(* Logix 5000 project; controller cal1615 1756-L62 rev 20.19; software revision 20.05; part 5 of 81 *)

        [6]   // Zone 1 Dint to HMI
        [6].0   // Zone 1 Dint to HMI Exhaut VFD Faulted
        [6].1   // Zone 1 Dint to HMI Exhaut VFD Warning
        [6].2   // Zone 1 Dint to HMI Exhaut VFD Running Forward
        [6].3   // Zone 1 Dint to HMI Exhaut VFD Running Reverse
        [6].4   // Zone 1 Dint to HMI Exhaut VFD Ready
        [6].5   // Zone 1 Dint to HMI Exhaut VFD Control from Net
        [6].6   // Zone 1 Dint to HMI Exhaut VFD Reference from Net
        [6].7   // Zone 1 Dint to HMI Exhaut VFD at Reference
        [6].8   // Zone 1 Dint to HMI Recirc VFD Faulted
        [6].9   // Zone 1 Dint to HMI Recirc VFD Warning
        [6].10   // Zone 1 Dint to HMI Recirc VFD Running Forward
        [6].11   // Zone 1 Dint to HMI Recirc VFD Running Reverse
        [6].12   // Zone 1 Dint to HMI Recirc VFD Ready
        [6].13   // Zone 1 Dint to HMI Recirc VFD Control from Net
        [6].14   // Zone 1 Dint to HMI Recirc VFD Reference from Net
        [6].15   // Zone 1 Dint to HMI Recirc VFD At Reference
        [6].16   // Zone 1 Dint to HMI Temperature Control PI: Request Heat
        [6].17   // Zone 1 Dint to HMI Temperature Control PI: Off
        [6].18   // Zone 1 Dint to HMI Temperature Control PI: Request Manual Control
        [6].19   // Zone 1 Dint to HMI Temperature Control PI:
        [6].20   // Zone 1 Dint to HMI PI:
        [6].21   // Zone 1 Dint to HMI PI:
        [6].22   // Zone 1 Dint to HMI PI:
        [6].23   // Zone 1 Dint to HMI PI:
        [6].24   // Zone 1 Dint to HMI PI:
        [6].25   // Zone 1 Dint to HMI PI:
        [6].26   // Zone 1 Dint to HMI PI:
        [6].27   // Zone 1 Dint to HMI PI:
        [6].28   // Zone 1 Dint to HMI PI:
        [6].29   // Zone 1 Dint to HMI PI:
        [6].30   // Zone 1 Dint to HMI PI:
        [6].31   // Zone 1 Dint to HMI PI:
        [7]   // Zone 1 Dint to HMI
        [8]   // Zone 1 Dint to HMI Temperature Control Status - State
        [9]   // Zone 1 Dint to HMI Temperature Control Status (Ready/Fault etc)
        [10]   // Zone 1 Dint to HMI Exhaust VFD Status
        [11]   // Zone 1 Dint to HMI Recirc VFD Status
        [12]   // Zone 1 Dint to HMI
        [13]   // Zone 1 Dint to HMI
        [14]   // Zone 1 Dint to HMI
        [15]   // Zone 1 Dint to HMI
   p11_do_enable_burner : BOOL := 1;   // Zone 1 Digital Output Enable Burner
   p11_do_exh : acs800_do_normal := (forward := 1);   // Zone 1 Digital Output Exhaust Fan
   p11_do_recirc : acs800_do_normal := (forward := 1);   // Zone 1 Digital Outputs Supply Fan
   p11_do_rst_flame : BOOL;   // Zone 1 Digital Output Reset Flame Safety
   p11_exhaust_input_max : REAL := 2000.0;
   p11_exhaust_input_min : REAL;   // Zone 1 Exhaust Input Minimum
   p11_exhaust_output_max : REAL := 2000.0;
   p11_exhaust_output_min : REAL;
   p11_hc_input_max : REAL := 100.0;
   p11_hc_input_min : REAL;
   p11_hc_output_max : REAL := 30840.0;
   p11_hc_output_min : REAL;
   p11_lfl_input_max : REAL := 30840.0;
   p11_lfl_input_min : REAL;
   p11_lfl_output_max : REAL := 100.0;
   p11_lfl_output_min : REAL;
   p11_param_fast_to_soak : REAL := 20.0;   // Zone 1 Parameter Fast to Soak Control
   p11_param_lfl_hhl : REAL := 40.0;   // Zone 1 Parameter High High Lower Flash Limit
   p11_param_lfl_hl : REAL := 25.0;   // Zone 1 Parameter High LFL Limit
   p11_param_pid1_ff : REAL := 25.0;   // Zone 1 Parameter Fast PID Bias
   p11_param_pid1_kd : REAL;   // Zone 1 Parameter Fast PID Derivative Gain
   p11_param_pid1_ki : REAL;   // Zone 1 Parameter Fast PID Integral Gain
   p11_param_pid1_kp : REAL := 50.0;   // Zone 1 Parameter Fast PID Proportional Gain
   p11_param_pid2_ff : REAL := 20.0;   // Zone 1 Parameter Auto PID Bias
   p11_param_pid2_kd : REAL;   // Zone 1 Parameter Auto PID Derivative Gain
   p11_param_pid2_ki : REAL := 1.0;   // Zone 1 Parameter Auto PID Integral Gain
   p11_param_pid2_kp : REAL := 20.0;   // Zone 1 Parameter Auto PID Proportional Gain
   p11_param_shutdown_temp : REAL := 110.0;   // Zone 1 Parameter Zone Shutdown Temperature
   p11_param_soak_to_fast : REAL := 20.0;   // Zone 1 Parameter Soak to Fast Control
   p11_param_tc01_dev : REAL := 20.0;   // Zone 1 Parameter Oven Temperature Deviation from Setpoint
   p11_param_tc01_hl : REAL := 440.0;   // Zone 1 Parameter Process Air High Limit
   p11_param_tc01z : REAL;   // Zone 1 Parameter Process Temperature Zero Offset
   p11_param_tc02z : REAL;   // Zone 1 Parameter SupplyTemperature Zero Offset
   p11_param_zone_pressure : REAL := -0.25;   // Zone 1 Parameter High Pressure LImit
   p11_prs_input_max : REAL := 30840.0;
   p11_prs_input_min : REAL;
   p11_prs_output_max : REAL := 0.25;
   p11_prs_output_min : REAL := -0.25;
   p11_real_to_hmi : REAL[112] := ([0] := 194.7, [1] := 194.7, [2] := 194.7, [6] := -0.25, [7] := 3.0804152, [8] := 30.891432, [9] := 4.9, [10] := 901.0, [12] := 37.748573, [13] := 22.2, [14] := 1101.0, [24] := 17.754694, [28] := 900.0, [30] := 1100.0, [44] := 50.0, [47] := 25.0, [48] := 20.0, [49] := 1.0, [51] := 20.0, [52] := 440.0, [54] := 20.0, [55] := 25.0, [56] := 40.0, [57] := 110.0, [58] := -0.25, [59] := 20.0, [60] := 20.0, [67] := 195.0, [68] := 45.0, [72] := 194.7);   // Zone 1 Real to HMI
        [0]   // Zone 1 Real to HMI Analog Input Zone 1 Process Control Temperature 1
        [1]   // Zone 1 Real to HMI Analog Input Zone 1 Process Control Temperature 2
        [2]   // Zone 1 Real to HMI Analog Input
        [3]   // Zone 1 Real to HMI Analog Input
        [6]   // Zone 1 Real to HMI Analog Input Pressure
        [7]   // Zone 1 Real to HMI Analog Input Lower Flash Limit
        [8]   // Zone 1 Real to HMI Analog Input Exhaust Fan Hz
        [9]   // Zone 1 Real to HMI Analog Input Exhaust Fan Amps
        [10]   // Zone 1 Real to HMI Analog Input Exhaust Fan RPM
        [11]   // Zone 1 Real to HMI Analog Input Exhaust Fan PCT
        [12]   // Zone 1 Real to HMI Analog Input Recirc Fan Hz
        [13]   // Zone 1 Real to HMI Analog Input Recirc Fan Amps
        [14]   // Zone 1 Real to HMI Analog Analog Input Recirc Fan RPM
        [15]   // Zone 1 Real to HMI Analog Analog Input Recirc Fan Pct
        [16]   // Zone 1 Real to HMI Analog Input Spare
        [17]   // Zone 1 Real to HMI Analog Input Spare
        [24]   // Zone 1 Real to HMI Analog Output Hot Air Damper
        [28]   // Zone 1 Real to HMI Analog Output Exhaust Fan VFD Selected Speed
        [30]   // Zone 1 Real to HMI Analog Output Supply Fan VFD Selected Speed
        [40]   // Zone 1 Real to HMI Parameter TC01 Temperature Zero Offset
        [41]   // Zone 1 Real to HMI Parameter TC02 Temperature Zero Offset
        [42]   // Zone 1 Real to HMI Parameter
        [43]   // Zone 1 Real to HMI Parameter
        [44]   // Zone 1 Real to HMI Parameter PID1 NKp
        [45]   // Zone 1 Real to HMI Parameter PID1 Ki
        [46]   // Zone 1 Real to HMI Parameter PID1 Kd
        [47]   // Zone 1 Real to HMI Parameter PID1 Bias
        [48]   // Zone 1 Real to HMI Parameter PID2 Kp
        [49]   // Zone 1 Real to HMI Parameter PID2 Ki
        [50]   // Zone 1 Real to HMI Parameter PID2 Kd
        [51]   // Zone 1 Real to HMI Parameter PID2 Bias
        [52]   // Zone 1 Real to HMI Parameter Process Control High Limit
        [53]   // Zone 1 Real to HMI Parameter Spare
        [54]   // Zone 1 Real to HMI parameter Process Control Deviation
        [55]   // Zone 1 Real to HMI Parameter LFL Warning Level
        [56]   // Zone 1 Real to HMI Parameter LFL Alarm Level
        [57]   // Zone 1 Real to HMI Parameter Zone Shutdown Temperature
        [58]   // Zone 1 Real to HMI Parameter High Pressure LImit
        [59]   // Zone 1 Real to HMI Temperature Control Fast to Soak Control Deviation
        [60]   // Zone 1 Real to HMI Temperature Control Soak to Fast Control Deviation
        [61]   // Zone 1 Real to HMI Parameter
        [62]   // Zone 1 Real to HMI Parameter
        [63]   // Zone 1 Real to HMI Parameter
        [64]   // Zone 1 Real to HMI Exhaust VFD RPM Setpoint
        [65]   // Zone 1 Real to HMI Recirc VFD RPM Setpoint
        [67]   // Zone 1 Real to HMI Temperature Control Setpoint
        [68]   // Zone 1 Real to HMI Temperature Control manual Control Valve Setpoint
        [69]   // Zone 1 Real to HMI
        [70]   // Zone 1 Real to HMI
        [71]   // Zone 1 Real to HMI
        [72]   // Zone 1 Real to HMI Process Control Temperature
        [73]   // Zone 1 Real to HMI
        [74]   // Zone 1 Real to HMI
        [75]   // Zone 1 Real to HMI
        [76]   // Zone 1 Real to HMI
        [77]   // Zone 1 Real to HMI
        [78]   // Zone 1 Real to HMI
        [79]   // Zone 1 Real to HMI
   p11_recirc_input_max : REAL := 2000.0;
   p11_recirc_input_min : REAL;
   p11_recirc_output_max : REAL := 2000.0;
   p11_recirc_output_min : REAL;
   p11r01 : routine := (comment := 7);   // Zone 1 Main
   p11r02 : routine := (comment := -1073741761);   // Zone 1 Misc Control
        .FAULT.0   // Zone 1 Misc Control
        .WARNING.0   // Zone 1 Misc Control Low Pressure
        .UNACK_FAULT   // Zone 1 Misc Control Unacknowledged Fault Exists
        .UNACK_WARNING   // Zone 1 Misc Control Unacknowledged Warning Exists
   p11r02_fault_exists : BOOL;
   p11r02_not_safe_temp : BOOL := 1;   // Zone 1 Misc Control Zone above Safe Temp
   p11r02_safe_temp : BOOL;   // Zone 1 Misc Control Zone Temperature at Safe Temp
   p11r02_shutdown_temp : BOOL;   // Zone 1 Misc Control Safe Shutdown Temperature
   p11r02_timer_fault : TIMER[4];   // Zone 1 Misc Control Fault Delay
   p11r02_timer_safe_temp : TIMER[2] := ([0].PRE := 30000, [1].PRE := 30000, [1].ACC := 30018, [1].EN := 1, [1].DN := 1);   // Zone 1 Misc Control Chamber SafeTemperature Dwell
   p11r02_timer_warning : TIMER[4] := ([0].PRE := 1500);   // Zone 1 Misc Control Warning Delay
   p11r02_unack_fault : BOOL;   // Zone 1 Misc Control Unacknowledged Fault Exists
   p11r02_unack_warning : BOOL;   // Zone 1 Misc Control Unacknowledged Warning Exists
   p11r02_warning_exists : BOOL := 1;
   p11r03 : routine := (comment := -1073741761);   // Zone 1 Input
        .UNACK_FAULT   // Zone 1 Input Unacknowledged Fault Exists
        .UNACK_WARNING   // Zone 1 Input Unacknowledged Warning Exists
   p11r03_hz : SYS_SCP := (Input := 901.0, Input_Max := 1750.0, Output_Max := 60.0, Output := 30.891432);   // Zone 1 Analog Inputs SCP Hz
   p11r03_timer_fault : TIMER[4];   // Zone 1 Input Fault Delay
   p11r03_timer_warning : TIMER[4];   // Zone 1 Input Warning Delay
   p11r04 : routine := (comment := -1073741761);   // Zone 1 Output
        .UNACK_FAULT   // Zone 1 Analog Output Unacknowledged Fault Exists
        .UNACK_WARNING   // Zone 1 Analog Output Unacknowledged Warning Exists
   p11r04_timer_fault : TIMER[4];   // Zone 1 Output Fault Delay
   p11r04_timer_warning : TIMER[4];   // Zone 1 Output Warning Delay
   p11r05 : routine := (comment := -1073741761, state := 7);   // Zone 1 Dint to HMI
        .UNACK_FAULT   // Zone 1 Dint to HMI Unacknowledged Fault Exists
        .UNACK_WARNING   // Zone 1 Dint to HMI Unacknowledged Warning Exists
   p11r05_exh_status : DINT := 2;
   p11r05_recirc_status : DINT := 2;
   p11r05_temp_ctrl_status : DINT := 2;
   p11r05_timer_fault : TIMER[4];   // Zone 1 Dint to HMI Fault Delay
   p11r05_timer_warning : TIMER[4];   // Zone 1 Dint to HMI Warning Delay
   p11r06 : routine := (comment := -1073741572);   // Zone 1 Real to HMI
        .UNACK_FAULT   // Zone 1 Real to HMI Unacknowledged Fault Exists
        .UNACK_WARNING   // Zone 1 Real to HMI Unacknowledged Warning Exists
   p11r06_timer_fault : TIMER[4];   // Zone 1 Real to HMI Fault Delay
   p11r06_timer_warning : TIMER[4];   // Zone 1 Real to HMI Warning Delay
   p11r07 : routine := (comment := -1073741761);   // Zone 1 Alarms
        .UNACK_FAULT   // Zone 1 Alarms Unacknowledged Fault Exists
        .UNACK_WARNING   // Zone 1 Alarms Unacknowledged Warning Exists
   p11r07_timer_fault : TIMER[4];   // Zone 1 Alarms Fault Delay
   p11r07_timer_warning : TIMER[4];   // Zone 1 Alarms Warning Delay
   p11r08 : routine := (comment := -1073741761);   // Zone 1 Warnings
        .UNACK_FAULT   // Zone 1 Warnings Unacknowledged Fault Exists
        .UNACK_WARNING   // Zone 1 Warnings Unacknowledged Warning Exists
   p11r08_timer_fault : TIMER[4];   // Zone 1 Warnings Fault Delay
   p11r08_timer_warning : TIMER[4];   // Zone 1 Warnings Warning Delay
   p11r09 : routine := (comment := -1073741761);   // Zone 1 Modes
        .FAULT.0   // Zone 1 Modes
        .UNACK_FAULT   // Zone 1 Modes Unacknowledged Fault Exists
        .UNACK_WARNING   // Zone 1 Modes Unacknowledged Warning Exists
   p11r09_timer_fault : TIMER[4];   // Zone 1 Modes Fault Delay
   p11r09_timer_warning : TIMER[8];   // Zone 1 Modes Warning Delay
   p11r10 : routine := (comment := -1073741761);   // Zone 1
        .UNACK_FAULT   // Zone 1 Parameters Unacknowledged Fault Exists
        .UNACK_WARNING   // Zone 1 Parameters Unacknowledged Warning Exists
   p11r10_timer_fault : TIMER[4];   // Zone 1 Fault Delay
   p11r10_timer_warning : TIMER[4];   // Zone 1 Warning Delay
   p11r12_Oven_auto_run_on : BOOL := 1;   // Zone 1 Temp Sequence Oven Auto Run On
   p11r16_pid_temp_cv : DINT := 16;   // Zone 1 Temperature Control Control Valve
   p11r16_temp_ok : BOOL := 1;   // Zone 1 Temperature Control Temperature OK
   p11r20 : routine := (comment := -1073741761);   // Zone 1 Temp Sequence
        .FAULT.0   // Zone 1
        .FAULT.1   // Zone 1
        .FAULT.2   // Zone 1
        .FAULT.3   // Zone 1
        .WARNING.0   // Zone 1
        .UNACK_FAULT   // Zone 1 Temp Sequence Unacknowledged Fault Exists
        .UNACK_WARNING   // Zone 1 Unacknowledged Warning Exists
   p11r20_safeties_ok : BOOL := 1;   // Zone 1 Temperature Control Burner Safeties OK this Lightoff
   p11r20_state : DINT := 1025;   // Zone 1 Temperature Control State
        .0   // Zone 1 Temperature Control State 0 One-Step per Scan
        .1   // Zone 1 Temperature Control State 1 Off
        .2   // Zone 1 Temperature Control State 2 Idle
        .3   // Zone 1 Temperature Control State 3 Start Recirculation Fan
        .4   // Zone 1 Temperature Control State 4 Start Exhaust Fan
        .5   // Zone 1 Temperature Control State 5 Wait for Safeties
        .6   // Zone 1 Temperature Control State 6 Safeties Made
        .7   // Zone 1 Temperature Control State 7 Purge
        .8   // Zone 1 Temperature Control State 8 Burner Lit
        .9   // Zone 1 Temperature Control State 9 Heat to Setpoint
        .10   // Zone 1 Temperature Control State 10 Control to Setpoint
        .11   // Zone 1 Temperature Control State 11 Cooldown
        .12   // Zone 1 Temperature Control State 12 Cooldown Fans
        .13   // Zone 1 Temperature Control State 13 Complete
        .31   // Zone 1 Temperature Control State 31 Manual
   p11r20_status : DINT := 10;   // Zone 1 Temperature Control Sequence Status
   p11r20_timer_fault : TIMER[4];   // Zone 1 Temp Sequence Fault Delay
   p11r20_timer_state_11 : TIMER := (PRE := 5000);   // Zone 1 Temp Sequence State 11 Dwell
   p11r20_timer_state_3 : TIMER := (PRE := 1000, ACC := 1022, EN := 1, DN := 1);   // Zone 1 Temperature Control State 3 Dwell
   p11r20_timer_state_4 : TIMER := (PRE := 1000, ACC := 1025, EN := 1, DN := 1);   // Zone 1 Temp Sequence State 4 Dwell
   p11r20_timer_state_7 : TIMER := (PRE := 2000, ACC := 2024, EN := 1, DN := 1);   // Zone 1 Temp Sequence State 7 Dwell
   p11r20_timer_warning : TIMER[4];   // Zone 1 Temp Sequence Warning Delay
   p11r30 : routine := (comment := -1073741697, oneshot := 4, warning := 192, warning_ack := 192);   // Zone 1 Temperature Control
        .FAULT.0   // Zone 1 Temperature Control Process Control Software High Limit
        .FAULT.1   // Zone 1 Temperature Control Process Control Hardware High Limit
        .FAULT.2   // Zone 1 Temperature Control Process Control Thermocouple Failure
        .FAULT.3   // Zone 1 Temperature Control Process Control Temperature Spare
        .FAULT.4   // Zone 1 Temperature Control Lower Flash Limit High High Limit Exceeded
        .FAULT.5   // Zone 1 Temperature Control Flame Failure
        .FAULT.6   // Zone 1 Temperature Control Burner Safeties Failure
        .FAULT.7   // Zone 1 Temperature Control Recirculation Fan Speed Fault
        .FAULT.8   // Zone 1 Temperature Control Exhaust Fan Speed Fault
        .FAULT.9   // Zone 1 Temperature Control Access Door Open
        .FAULT.10   // Zone 1 Temperature Control Spare
        .FAULT.11   // Zone 1 Temperature Control
        .FAULT.12   // Zone 1 Temperature Control Spare
        .FAULT.13   // Zone 1 Temperature Control
        .FAULT.14   // Zone 1 Temperature Control
        .WARNING.0   // Zone 1 Temperature Control Control Temperature Deviation
        .WARNING.1   // Zone 1 Temperature Control Process Control Thermocouple 1 Failure
        .WARNING.2   // Zone 1 Temperature Control Process Control Thermocouple 2 Failure
        .WARNING.3   // Zone 1 Temperature Control Control Valve in Manual
        .WARNING.4   // Zone 1 Temperature Control LFL High Limit
        .WARNING.5   // Zone 1 Temperature Control Zone Off
        .WARNING.6   // Zone 1 Temperature Control Fresh Air Filter Dirty
        .WARNING.7   // Zone 1 Temperature Control Combustion Air Filter Dirty
        .WARNING.8   // Zone 1 Temperature Control Recirculation Air Filter Dirty
        .UNACK_FAULT   // Zone 1 Temperature Control Unacknowledged Fault Exists
        .UNACK_WARNING   // Zone 1 Temperature Control Unacknowledged Warning Exists
   p11r30_cv_man_sp : REAL := 45.0;   // Zone 1 Temperature Control Manual Heat Control Valve Setpoint
   p11r30_pb_auto : BOOL;   // Zone 1 Temperature Control PB: Zone Control Auto
   p11r30_pb_manual : BOOL;   // Zone 1 Temperature Control PB: Zone Control Manual
   p11r30_pb_zone_off : BOOL;   // Zone 1 Temperature Control PB: Stop Zone Heat Control
   p11r30_pb_zone_on : BOOL;   // Zone 1 Temperature Control PB: Start Zone Heat Control
   p11r30_permissive_run : BOOL := 1;   // Zone 1 Temperature Control Run Permissive
   p11r30_pid_temp : PID := (CTL := -2144304000, EN := 1, NOBC := 1, NOZC := 1, INI := 1, DVNA := 1, PVHA := 1, SP := 195.0, KP := 20.0, KI := 1.0, BIAS := 20.0, MAXS := 1000.0, SO := 16.278357, MAXO := 100.0, UPD := 0.01, PV := 195.40001, ERR := -0.40000916, OUT := 16.278357, MAXI := 10000.0, MAXCV := 100.0, MAXTIE := 100.0, DATA[0] := -2.9216259, DATA[1] := -312.64, DATA[2] := 195.40001, DATA[3] := -0.40000916, DATA[4] := 195.0, DATA[5] := 0.1, DATA[6] := 0.1, DATA[7] := 0.16, DATA[8] := 20.0, DATA[9] := 1.0, DATA[11] := 20.0, DATA[12] := 1.0, DATA[15] := 1.0, DATA[16] := 1.0);   // Zone 1 Temperature Control PID
   p11r30_pid_temp_pv : REAL := 1954.0001;   // Zone 1 Temperature Control PID Temp Process Variable
   p11r30_pid_temp_sp : REAL := 195.0;   // Zone 1 Temperature Control PID Temperature Control Setpoint
   p11r30_pid_temp_sp_error : REAL := 0.40000916;   // Zone 1 Temperature Control Setpoint/Process Variable Error (ABS)
   p11r30_pid_temp_sp_last : REAL := 195.0;   // Zone 1 Temperature Control Setpoint Last Scan
   p11r30_request_deviation_warning : BOOL := 1;   // Zone 1 Temperature Control Request Setpoint Deviation Warning
   p11r30_request_heat : BOOL := 1;   // Zone 1 Temperature Control Request Heat
   p11r30_request_heat_last : BOOL := 1;   // Zone 1 Temperature Control Request Heat Last Scan
   p11r30_request_manual : BOOL;   // Zone 1 Temperature Control Request Manual Control
   p11r30_request_PID_shot : BOOL;
   p11r30_request_soak_control : BOOL := 1;   // Zone 1 Temperature Control Request Soak Control
   p11r30_temp_deviation_setpoint : DINT := 5;
   p11r30_timer_fault : TIMER[16] := ([0].PRE := 5000, [2].PRE := 1000, [4].PRE := 1000, [10].PRE := 5000, [11].PRE := 5000, [12].PRE := 5000);   // Zone 1 Temperature Control Fault Delay
   p11r30_timer_warning : TIMER[12] := ([0].PRE := 10000, [1].PRE := 1000, [2].PRE := 1000, [3].PRE := 90000, [4].PRE := 1000, [6].PRE := 1000, [6].ACC := 1023, [6].EN := 1, [6].DN := 1, [7].PRE := 1000, [7].ACC := 1031, [7].EN := 1, [7].DN := 1, [8].PRE := 1000);   // Zone 1 Temperature Control Warning Delay
   p11r30_vfds_ok : BOOL := 1;
   p11r30_vfds_ready : BOOL := 1;   // Zone 1 Temperature Control VFDs On
   p11r31 : routine := (comment := -1073741697);   // Zone 1 Exhaust VFD
        .FAULT.0   // Zone 1 Exhaust VFD Drive Fault
        .FAULT.1   // Zone 1 Exhaust VFD Motor Thermistor Not OK
        .FAULT.2   // Zone 1 Exhaust VFD Not Ready
        .FAULT.3   // Zone 1 Exhaust VFD
        .WARNING.0   // Zone 1 Exhaust VFD VFD Stopped While Chamber is Too Hot
        .WARNING.1   // Zone 1 Exhaust VFD Fan Flow Failure
        .WARNING.2   // Zone 1 Exhaust VFD VFD Warning
        .UNACK_FAULT   // Zone 1 Exhaust VFD Unacknowledged Fault Exists
        .UNACK_WARNING   // Zone 1 Exhaust VFD Unacknowledged Warning Exists
   p11r31_pb_start : BOOL;   // Zone 1 Exhaust VFD PB: Start
   p11r31_pb_stop : BOOL;   // Zone 1 Exhaust VFD PB: Stop
   p11r31_request_auto_run : BOOL := 1;   // Zone 1 Exhaust Fan Run Request
   p11r31_request_auto_stop : BOOL := 1;   // Zone 1 Exhaust VFD Request Auto Stop
   p11r31_run_permissive : BOOL := 1;   // Zone 1 Exhaust VFD Run Permissive
   p11r31_timer_fault : TIMER[5] := ([1].PRE := 500);   // Zone 1 Exhaust VFD Fault Timer
   p11r31_timer_prs : TIMER := (PRE := 2500);   // Advanced Cooling Pump Pressure On Delay
   p11r31_timer_warning : TIMER[5] := ([0].PRE := 10000, [1].PRE := 20000, [2].PRE := 500);   // Zone 1 Exhaust VFD Waringing Timer
   p11r31_vfd_stopped : BOOL;   // Zone 1 Exhaust VFD VFD Stopped
   p11r32 : routine := (comment := -536870849);   // Zone 1 Recirc VFD
        .FAULT.0   // Zone 1 Recirc VFD Drive Fault
        .FAULT.1   // Zone 1 Recirc VFD Motor Thermistor Not OK
        .FAULT.2   // Zone 1 Recirc VFD Not Ready
        .FAULT.3   // Zone 1 Supply VFD
        .WARNING.0   // Zone 1 Recirc VFD VFD Stopped While Chamber is Too Hot
        .WARNING.1   // Zone 1 Recirc VFD Fan Flow Failure
        .WARNING.2   // Zone 1 Recirc VFD VFD Warning
        .UNACK_FAULT   // Zone 1 Recirc VFD Unacknowledged Fault Exists
        .UNACK_WARNING   // Zone 1 Recirc VFD Unacknowledged Warning Exists
   p11r32_pb_start : BOOL;   // Zone 1 Recirc VFD PB: Start
   p11r32_pb_stop : BOOL;   // Zone 1 Recirc VFD PB: Stop
   p11r32_request_auto_run : BOOL := 1;   // Zone 1 Recirc Fan Run Request
   p11r32_request_auto_stop : BOOL := 1;   // Zone 1 Recirc VFD Request Auto Stop
   p11r32_run_permissive : BOOL := 1;   // Zone 1 Recirc VFD Run Permissive
   p11r32_timer_fault : TIMER[5] := ([1].PRE := 500);   // Zone 1 Recirc VFD Fault Timer
   p11r32_timer_warning : TIMER[5] := ([0].PRE := 10000, [1].PRE := 20000, [2].PRE := 20000);   // Zone 1 Supply VFD Warning Timer
   p11r32_vfd_stopped : BOOL;   // Zone 1 Recirc VFD VFD Stopped
   p12_ai_exhaust_amps : REAL := 2.2;   // Zone 2 Analog Input Exhaust Fan Amps
   p12_ai_exhaust_hz : REAL := 30.891432;   // Zone 2 Analog Input Exhaust Fan HZ
   p12_ai_exhaust_hz_max : REAL := 60.0;   // Zone 2 Analog Input Exhaust Fan Max HZ
   p12_ai_exhaust_pct : REAL;   // Zone 2 Analog Input Exhaust Fan PCT
   p12_ai_exhaust_rpm : REAL := 901.0;   // Zone 2 Analog Input Exhaust Fan RPM
   p12_ai_lfl : REAL;   // Zone 2 Analog Input Lower Flash Limit
   p12_ai_prs : REAL := -0.0545042;   // Zone 2 Analog Input Pressure
   p12_ai_recirc_amps : REAL;   // Zone 2 Analog Input Recirc Fan Amps
   p12_ai_recirc_hz : REAL;   // Zone 2 Analog Input Supply Fan HZ
   p12_ai_recirc_hz_max : REAL;   // Zone 2 Analog Input Supply Fan Max HZ
   p12_ai_recirc_pct : REAL;   // Zone 2 Analog Input Recirc Fan PCT
   p12_ai_recirc_rpm : REAL := 1100.0;   // Zone 2 Analog Input Recirc Fan RPM
   p12_ai_tc01 : REAL := 199.40001;   // Zone 2 Analog Input Control Thermocouple 1
   p12_ai_tc02 : REAL := 199.7;   // Zone 2 Analog Input Control Thermocouple 2
   p12_ao_cv : REAL := 27.222637;   // Zone 2 Analog Output Control Valve
   p12_ao_exhaust_selected_speed : REAL := 900.0;   // Zone 2 Analog Output Exhaust Fan VFD Selected Speed
   p12_ao_recirc_selected_speed : REAL := 1100.0;   // Zone 2 Analog Output Recirc Fan VFD Selected Speed
   p12_di_burner_auto : BOOL := 1;   // Zone 2 Digital Input Burner Auto
   p12_di_burner_safeties_ok : BOOL := 1;   // Zone 2 Digital Input Burner Safeties Ok
   p12_di_door_open : BOOL;   // Zone 2 Digital Input Access Door Open
   p12_di_exh : acs800_di_normal := (running_fwd := 1, ready := 1, ctrl_from_net := 1, ref_from_net := 1, at_reference := 1);   // Zone 2 Digital Inputs Exhaust Fan
        .FAULTED   // Zone 2 Digital Inputs Exhaust Fan
   p12_di_exh_fan_mtr_ts : BOOL := 1;   // Zone 2 Digital Input Exhaust Fan Motor Thermostat OK
   p12_di_exh_flow_ok : BOOL := 1;   // Zone 2 Digital Input Exhaust Flow OK
   p12_di_flame_failure : BOOL;   // Zone 2 Digital Input Flame Failure
   p12_di_flame_on : BOOL := 1;   // Zone 2 Digital Input Burner is On
   p12_di_fresh_air_clean : BOOL;   // Zone 2 Digital Input Fresh Air Filter Dirty
   p12_di_high_limit_temp_ok : BOOL := 1;   // Zone 2 Digital Input High Limit Temperature OK
   p12_di_recirc : acs800_di_normal := (running_fwd := 1, ready := 1, ctrl_from_net := 1, ref_from_net := 1, at_reference := 1);   // Zone 2 Digital Inputs Recirc Fan
   p12_di_recirc_fan_mtr_ts : BOOL := 1;   // Zone 2 Digital Input Recirc Fan Motor Thermostat OK
   p12_di_recirc_flow_ok : BOOL := 1;   // Zone 2 Digital Input Recirc Flow OK
   p12_di_sp0 : BOOL;
   p12_di_sp00 : BOOL;   // Zone 2 Digital Input Combustion Blower Pressure OK
   p12_di_sp1 : BOOL;
   p12_di_sp2 : BOOL;
   p12_di_sp3 : BOOL;
   p12_di_tc01_bo : BOOL;   // Zone 2 Digital Input Control Thermocouple 1 Failure
   p12_di_tc02_bo : BOOL;   // Zone 2 Digital Input Control Thermocouple 2 Failure
   p12_di_zone_air_clean : BOOL;   // Zone 2 Digital Input Zone 2 Filter Dirty
   p12_dint_to_hmi : DINT[16] := ([2] := 192, [4] := 591187, [5] := 50532323, [6] := 62708, [8] := 10, [9] := 2, [10] := 2, [11] := 2);   // Zone 2 Temperature Control VFDs On
        [0]   // Zone 2 Dint to HMI Alarms
        [0].0   // Zone 2 Dint to HMI Alarms A00: Process Control Software High Limit
        [0].1   // Zone 2 Dint to HMI Alarms A01: Process Control Hardware High Limit
        [0].2   // Zone 2 Dint to HMI Alarms A02: Process Control Thermocouple Failure
        [0].3   // Zone 2 Dint to HMI Alarms A03: Process Control Temperature Spare
        [0].4   // Zone 2 Dint to HMI Alarms A04: Lower Flash Limit High High Limit Exceeded
        [0].5   // Zone 2 Dint to HMI Alarms A05: Flame Failure
        [0].6   // Zone 2 Dint to HMI Alarms A06: Burner Safeties Failure
        [0].7   // Zone 2 Dint to HMI Alarms A07: Recirculation Fan Speed Fault
        [0].8   // Zone 2 Dint to HMI Alarms A08: Exhaust Fan Speed Fault
        [0].9   // Zone 2 Dint to HMI Alarms A09: Access Door Open
        [0].10   // Zone 2 Dint to HMI Alarms A10:
        [0].11   // Zone 2 Dint to HMI Alarms A11:
        [0].12   // Zone 2 Dint to HMI Alarms A12:
        [0].13   // Zone 2 Dint to HMI Alarms A13:
        [0].14   // Zone 2 Dint to HMI Alarms A14:
        [0].15   // Zone 2 Dint to HMI Alarms A15:
        [0].16   // Zone 2 Dint to HMI Alarms A16: Exhaust Fan Drive Fault
        [0].17   // Zone 2 Dint to HMI Alarms A17: Exhaust Fan Motor Thermistor Not OK
        [0].18   // Zone 2 Dint to HMI Alarms A18: Exhaust Fan VFD Not Ready
        [0].19   // Zone 2 Dint to HMI Alarms A19:
        [0].20   // Zone 2 Dint to HMI Alarms A20: Recirculation Fan Drive Fault
        [0].21   // Zone 2 Dint to HMI Alarms A21: Recirculation Fan Motor Thermistor Not OK
        [0].22   // Zone 2 Dint to HMI Alarms A22: Recirculation Fan VFD Not Ready
        [0].23   // Zone 2 Dint to HMI Alarms A23:
        [0].24   // Zone 2 Dint to HMI Alarms A24:
        [0].25   // Zone 2 Dint to HMI Alarms A25:
        [0].26   // Zone 2 Dint to HMI Alarms A26:
        [0].27   // Zone 2 Dint to HMI Alarms A27:
        [0].28   // Zone 2 Dint to HMI Alarms A28:
        [0].29   // Zone 2 Dint to HMI Alarms A29:
        [0].30   // Zone 2 Dint to HMI Alarms A30:
        [0].31   // Zone 2 Dint to HMI Alarms A31:
        [1]   // Zone 2 Dint to HMI Alarms
        [1].0   // Zone 2 Dint to HMI Alarms
        [1].1   // Zone 2 Dint to HMI Alarms
        [1].2   // Zone 2 Dint to HMI Alarms
        [1].3   // Zone 2 Dint to HMI Alarms
        [1].4   // Zone 2 Dint to HMI Alarms
        [1].5   // Zone 2 Dint to HMI Alarms
        [1].6   // Zone 2 Dint to HMI Alarms
        [1].7   // Zone 2 Dint to HMI Alarms
        [1].8   // Zone 2 Dint to HMI Alarms
        [1].9   // Zone 2 Dint to HMI Alarms
        [1].10   // Zone 2 Dint to HMI Alarms
        [1].11   // Zone 2 Dint to HMI Alarms
        [1].12   // Zone 2 Dint to HMI Alarms
        [1].13   // Zone 2 Dint to HMI Alarms
        [1].14   // Zone 2 Dint to HMI Alarms
        [1].15   // Zone 2 Dint to HMI Alarms
        [1].16   // Zone 2 Dint to HMI Alarms
        [1].17   // Zone 2 Dint to HMI Alarms
        [1].18   // Zone 2 Dint to HMI Alarms
        [1].19   // Zone 2 Dint to HMI Alarms
        [1].20   // Zone 2 Dint to HMI Alarms
        [1].21   // Zone 2 Dint to HMI Alarms
        [1].22   // Zone 2 Dint to HMI Alarms
        [1].23   // Zone 2 Dint to HMI Alarms
        [1].24   // Zone 2 Dint to HMI Alarms
        [1].25   // Zone 2 Dint to HMI Alarms
        [1].26   // Zone 2 Dint to HMI Alarms
        [1].27   // Zone 2 Dint to HMI Alarms
        [1].28   // Zone 2 Dint to HMI Alarms
        [1].29   // Zone 2 Dint to HMI Alarms
        [1].30   // Zone 2 Dint to HMI Alarms
        [1].31   // Zone 2 Dint to HMI Alarms
        [2]   // Zone 2 Dint to HMI Warnings
        [2].0   // Zone 2 Dint to HMI Warnings W00: Control Temperature Deviation
        [2].1   // Zone 2 Dint to HMI Warnings W01: Process Control Thermocouple 1 Failure
        [2].2   // Zone 2 Dint to HMI Warnings W02: Process Control Thermocouple 2 Failure
        [2].3   // Zone 2 Dint to HMI Warnings W03: Control Valve in Manual
        [2].4   // Zone 2 Dint to HMI Warnings W04: LFL High Limit
        [2].5   // Zone 2 Dint to HMI Warnings W05:
        [2].6   // Zone 2 Dint to HMI Warnings W06: Fresh Air Filter Dirty
        [2].7   // Zone 2 Dint to HMI Warnings W07: Combustion Air Filter Dirty
        [2].8   // Zone 2 Dint to HMI Warnings W08: Recirculation Air Filter Dirty
        [2].9   // Zone 2 Dint to HMI Warnings W09:
        [2].10   // Zone 2 Dint to HMI Warnings W10:
        [2].11   // Zone 2 Dint to HMI Warnings W11:
        [2].12   // Zone 2 Dint to HMI Warnings W12:
        [2].13   // Zone 2 Dint to HMI Warnings W13:
        [2].14   // Zone 2 Dint to HMI Warnings W14:
        [2].15   // Zone 2 Dint to HMI Warnings W15: Low Pressure
        [2].16   // Zone 2 Dint to HMI Warnings W16: Exhaust Fan Stopped While Zone is Too Hot
        [2].17   // Zone 2 Dint to HMI Warnings W17:
        [2].18   // Zone 2 Dint to HMI Warnings W18:
        [2].19   // Zone 2 Dint to HMI Warnings W19:
        [2].20   // Zone 2 Dint to HMI Warnings W20: Recirculation Fan Stopped While Zone is Too Hot
        [2].21   // Zone 2 Dint to HMI Warnings W21: Recirculation Fan Flow Failure
        [2].22   // Zone 2 Dint to HMI Warnings W22: Recirculation Fan Pressure Failure
        [2].23   // Zone 2 Dint to HMI Warnings W23:
        [2].24   // Zone 2 Dint to HMI Warnings W24:
        [2].25   // Zone 2 Dint to HMI Warnings W25:
        [2].26   // Zone 2 Dint to HMI Warnings W26:
        [2].27   // Zone 2 Dint to HMI Warnings W27:
        [2].28   // Zone 2 Dint to HMI Warnings W28:
        [2].29   // Zone 2 Dint to HMI Warnings W29:
        [2].30   // Zone 2 Dint to HMI Warnings W30:
        [2].31   // Zone 2 Dint to HMI Warnings W31:
        [3]   // Zone 2 Dint to HMI Warnings
        [3].0   // Zone 2 Dint to HMI Alarms
        [3].1   // Zone 2 Dint to HMI Alarms
        [3].2   // Zone 2 Dint to HMI Alarms
        [3].3   // Zone 2 Dint to HMI Alarms
        [3].4   // Zone 2 Dint to HMI Alarms
        [3].5   // Zone 2 Dint to HMI Alarms
        [3].6   // Zone 2 Dint to HMI Alarms
        [3].7   // Zone 2 Dint to HMI Alarms
        [3].8   // Zone 2 Dint to HMI Alarms
        [3].9   // Zone 2 Dint to HMI Alarms
        [3].10   // Zone 2 Dint to HMI Alarms
        [3].11   // Zone 2 Dint to HMI Alarms
        [3].12   // Zone 2 Dint to HMI Alarms
        [3].13   // Zone 2 Dint to HMI Alarms
        [3].14   // Zone 2 Dint to HMI Alarms
        [3].15   // Zone 2 Dint to HMI Alarms
        [3].16   // Zone 2 Dint to HMI Alarms
        [3].17   // Zone 2 Dint to HMI Alarms
        [3].18   // Zone 2 Dint to HMI Alarms
        [3].19   // Zone 2 Dint to HMI Alarms
        [3].20   // Zone 2 Dint to HMI Alarms
        [3].21   // Zone 2 Dint to HMI Alarms
        [3].22   // Zone 2 Dint to HMI Alarms
        [3].23   // Zone 2 Dint to HMI Alarms
        [3].24   // Zone 2 Dint to HMI Alarms
        [3].25   // Zone 2 Dint to HMI Alarms
        [3].26   // Zone 2 Dint to HMI Alarms
        [3].27   // Zone 2 Dint to HMI Alarms
        [3].28   // Zone 2 Dint to HMI Alarms
        [3].29   // Zone 2 Dint to HMI Alarms
        [3].30   // Zone 2 Dint to HMI Alarms
        [3].31   // Zone 2 Dint to HMI Alarms
        [4]   // Zone 2 Dint to HMI Process Indicators
        [4].0   // Zone 2 Dint to HMI PI: Zone Fault
        [4].1   // Zone 2 Dint to HMI PI: VFDs On/Ready
        [4].2   // Zone 2 Dint to HMI PI:
        [4].3   // Zone 2 Dint to HMI PI:
        [4].4   // Zone 2 Dint to HMI Exhaust VFD PI: Request Auto Run
        [4].5   // Zone 2 Dint to HMI Exhaust VFD PI: VFD Stopped
        [4].6   // Zone 2 Dint to HMI Exhaust VFD PI: Request Auto Stop
        [4].7   // Zone 2 Dint to HMI Exhaust VFD PI:
        [4].8   // Zone 2 Dint to HMI Recirc VFD PI: Request Auto Run
        [4].9   // Zone 2 Dint to HMI Recirc VFD PI: VFD Stopped
        [4].10   // Zone 2 Dint to HMI Recirc VFD PI: Request Auto Stop
        [4].11   // Zone 2 Dint to HMI Supply VFD PI:
        [4].12   // Zone 2 Dint to HMI PI:
        [4].13   // Zone 2 Dint to HMI PI:
        [4].14   // Zone 2 Dint to HMI PI:
        [4].15   // Zone 2 Dint to HMI PI:
        [4].16   // Zone 2 Dint to HMI Temperature Control PI: Request Heat
        [4].17   // Zone 2 Dint to HMI Temperature Control PI: Off
        [4].18   // Zone 2 Dint to HMI Temperature Control PI: Request Manual Control
        [4].19   // Zone 2 Dint to HMI Temperature Control PI: Request Auto Control
        [4].20   // Zone 2 Dint to HMI PI:
        [4].21   // Zone 2 Dint to HMI PI:
        [4].22   // Zone 2 Dint to HMI PI:
        [4].23   // Zone 2 Dint to HMI PI:
        [4].24   // Zone 2 Dint to HMI PI:
        [4].25   // Zone 2 Dint to HMI PI:
        [4].26   // Zone 2 Dint to HMI PI:
        [4].27   // Zone 2 Dint to HMI PI:
        [4].28   // Zone 2 Dint to HMI PI:
        [4].29   // Zone 2 Dint to HMI PI:
        [4].30   // Zone 2 Dint to HMI PI:
        [4].31   // Zone 2 Dint to HMI PI:
        [5]   // Zone 2 Dint to HMI Process Indicators
        [5].0   // Zone 2 Dint to HMI PI: Digital Input Burner Auto
        [5].1   // Zone 2 Dint to HMI PI: Digital Input Burner Safeties Ok
        [5].2   // Zone 2 Dint to HMI PI: Digital Input Combustion Air Filter Clean
        [5].3   // Zone 2 Dint to HMI PI: Digital Input Combustion Blower Pressure OK
        [5].4   // Zone 2 Dint to HMI PI: Digital Input Access Door Open
        [5].5   // Zone 2 Dint to HMI PI: Digital Input Exhaust Fan Motor Thermostat OK
        [5].6   // Zone 2 Dint to HMI PI: Digital Input Exhaust Flow OK
        [5].7   // Zone 2 Dint to HMI PI: Digital Input Flame Failure
        [5].8   // Zone 2 Dint to HMI PI: Digital Input Burner is On
        [5].9   // Zone 2 Dint to HMI PI: Digital Input High Limit Temperature OK
        [5].10   // Zone 2 Dint to HMI PI: Digital Input Recirc Fan Motor Thermostat OK
        [5].11   // Zone 2 Dint to HMI PI: Digital Input Recirc Flow OK
        [5].12   // Zone 2 Dint to HMI PI: Digital Input Recirculation Air Filter Clean
        [5].13   // Zone 2 Dint to HMI PI: Digital Input Fresh Air Filter Clean
        [5].14   // Zone 2 Dint to HMI PI: Digital Input Control Thermocouple 1 Failure
        [5].15   // Zone 2 Dint to HMI PI: Digital Input Control Thermocouple 2 Failure
        [6]   // Zone 2 Dint to HMI
        [6].0   // Zone 2 Dint to HMI Exhaust Fan Faulted
        [6].1   // Zone 2 Dint to HMI Exhaust Fan Warning
        [6].2   // Zone 2 Dint to HMI Exhaust Fan Running Forward
        [6].3   // Zone 2 Dint to HMI Exhaust Fan Running Reverse
        [6].4   // Zone 2 Dint to HMI Exhaust Fan Ready
        [6].5   // Zone 2 Dint to HMI Exhaust Fan Control from Net
        [6].6   // Zone 2 Dint to HMI Exhaust Fan Reference from Net
        [6].7   // Zone 2 Dint to HMI Exhaust Fan At Reference
        [6].8   // Zone 2 Dint to HMI Recirc Fan Faulted
        [6].9   // Zone 2 Dint to HMI Recirc Fan Warning
        [6].10   // Zone 2 Dint to HMI Recirc Fan Running Forward
        [6].11   // Zone 2 Dint to HMI Recirc Fan Running Reverse
        [6].12   // Zone 2 Dint to HMI Recirc Fan Ready
        [6].13   // Zone 2 Dint to HMI Recirc Fan Control from Net
        [6].14   // Zone 2 Dint to HMI Recirc Fan Reference from Net
        [6].15   // Zone 2 Dint to HMI Recirc Fan At Reference
        [6].16   // Zone 2 Dint to HMI Temperature Control PI: Request Heat
        [6].17   // Zone 2 Dint to HMI Temperature Control PI: Off
        [6].18   // Zone 2 Dint to HMI Temperature Control PI: Request Manual Control
        [6].19   // Zone 2 Dint to HMI Temperature Control PI:
        [6].20   // Zone 2 Dint to HMI PI:
        [6].21   // Zone 2 Dint to HMI PI:
        [6].22   // Zone 2 Dint to HMI PI:
        [6].23   // Zone 2 Dint to HMI PI:
        [6].24   // Zone 2 Dint to HMI PI:
        [6].25   // Zone 2 Dint to HMI PI:
        [6].26   // Zone 2 Dint to HMI PI:
        [6].27   // Zone 2 Dint to HMI PI:
        [6].28   // Zone 2 Dint to HMI PI:
        [6].29   // Zone 2 Dint to HMI PI:
        [6].30   // Zone 2 Dint to HMI PI:
        [6].31   // Zone 2 Dint to HMI PI:
        [7]   // Zone 2 Dint to HMI
        [8]   // Zone 2 Dint to HMI Temperature Control Status - State
        [9]   // Zone 2 Dint to HMI Temperature Control Status (Ready/Fault etc)
        [10]   // Zone 2 Dint to HMI Exhaust VFD Status
        [11]   // Zone 2 Dint to HMI Recirc VFD Status
        [12]   // Zone 2 Dint to HMI
        [13]   // Zone 2 Dint to HMI
        [14]   // Zone 2 Dint to HMI
        [15]   // Zone 2 Dint to HMI
   p12_do_enable_burner : BOOL := 1;   // Zone 2 Digital Output Enable Burner
   p12_do_exh : acs800_do_normal := (forward := 1);   // Zone 2 Digital Output Exhaust Fan
   p12_do_recirc : acs800_do_normal := (forward := 1);   // Zone 2 Digital Outputs Supply Fan
   p12_do_rst_flame : BOOL;   // Zone 2 Digital Output Reset Flame Safety
   p12_exhaust_input_max : REAL := 2000.0;
   p12_exhaust_input_min : REAL;
   p12_exhaust_output_max : REAL := 2000.0;
   p12_exhaust_output_min : REAL;
   p12_hc_input_max : REAL := 100.0;
   p12_hc_input_min : REAL;
   p12_hc_output_max : REAL := 30840.0;
   p12_hc_output_min : REAL;
   p12_lfl_input_max : REAL := 30840.0;
   p12_lfl_input_min : REAL;
   p12_lfl_output_max : REAL := 100.0;
   p12_lfl_output_min : REAL;
   p12_param_fast_to_soak : REAL := 5.0;   // Zone 2 Parameter Fast to Soak Control
   p12_param_lfl_hhl : REAL := 40.0;   // Zone 2 Parameter High High Lower Flash Limit
   p12_param_lfl_hl : REAL := 25.0;   // Zone 2 Parameter High LFL Limit
   p12_param_pid1_ff : REAL := 25.0;   // Zone 2 Parameter Fast PID Bias
   p12_param_pid1_kd : REAL;   // Zone 2 Parameter Fast PID Derivative Gain
   p12_param_pid1_ki : REAL;   // Zone 2 Parameter Fast PID Integral Gain
   p12_param_pid1_kp : REAL := 50.0;   // Zone 2 Parameter Fast PID Proportional Gain
   p12_param_pid2_ff : REAL := 15.0;   // Zone 2 Parameter Auto PID Bias
   p12_param_pid2_kd : REAL;   // Zone 2 Parameter Auto PID Derivative Gain
   p12_param_pid2_ki : REAL := 0.5;   // Zone 2 Parameter Auto PID Integral Gain
   p12_param_pid2_kp : REAL := 20.0;   // Zone 2 Parameter Auto PID Proportional Gain
   p12_param_shutdown_temp : REAL := 122.0;   // Zone 2 Parameter Zone Shutdown Temperature
   p12_param_soak_to_fast : REAL := 15.0;   // Zone 2 Parameter Soak to Fast Control
   p12_param_tc01_dev : REAL := 20.0;   // Zone 2 Parameter Oven Temperature Deviation from Setpoint
   p12_param_tc01_hl : REAL := 440.0;   // Zone 2 Parameter Process Air High Limit
   p12_param_tc01z : REAL;   // Zone 2 Parameter Process Temperature Zero Offset
   p12_param_tc02z : REAL;   // Zone 2 Parameter SupplyTemperature Zero Offset
   p12_param_zone_pressure : REAL := -0.25;   // Zone 2 Parameter High Pressure LImit
   p12_prs_input_max : REAL := 30860.0;
   p12_prs_input_min : REAL;
   p12_prs_output_max : REAL := 0.25;
   p12_prs_output_min : REAL := -0.25;
   p12_real_to_hmi : REAL[112] := ([0] := 199.5, [1] := 199.7, [2] := 199.5, [6] := -0.05241412, [8] := 30.891432, [9] := 2.2, [10] := 901.0, [14] := 1100.0, [24] := 27.046467, [28] := 900.0, [30] := 1100.0, [44] := 50.0, [47] := 25.0, [48] := 20.0, [49] := 0.5, [51] := 15.0, [52] := 440.0, [54] := 20.0, [55] := 25.0, [56] := 40.0, [57] := 122.0, [58] := -0.25, [59] := 5.0, [60] := 15.0, [67] := 200.0, [68] := 60.0, [72] := 199.5);   // Zone 2 Real to HMI
        [0]   // Zone 2 Real to HMI Analog Input Zone 2 Process Control Temperature 1
        [1]   // Zone 2 Real to HMI Analog Input Zone 2 Process Control Temperature 2
        [2]   // Zone 2 Real to HMI Analog Input
        [3]   // Zone 2 Real to HMI Analog Input
        [6]   // Zone 2 Real to HMI Analog Input Pressure
        [7]   // Zone 2 Real to HMI Analog Input Lower Flash Limit
        [8]   // Zone 2 Real to HMI Analog Input Exhaust Fan Hz
        [9]   // Zone 2 Real to HMI Analog Input Exhaust Fan Amps
        [10]   // Zone 2 Real to HMI Analog Input Exhaust Fan RPM
        [11]   // Zone 2 Real to HMI Analog Input Exhaust Fan PCT
        [12]   // Zone 2 Real to HMI Analog Input Recirc Fan Hz
        [13]   // Zone 2 Real to HMI Analog Input Recirc Fan Amps
        [14]   // Zone 2 Real to HMI Analog Analog Input Recirc Fan RPM
        [15]   // Zone 2 Real to HMI Analog Analog Input Recirc Fan Pct
        [16]   // Zone 2 Real to HMI Analog Input Spare
        [17]   // Zone 2 Real to HMI Analog Input Spare
        [24]   // Zone 2 Real to HMI Analog Output Hot Air Damper
        [28]   // Zone 2 Real to HMI Analog Output Exhaust Fan VFD Selected Speed
        [30]   // Zone 2 Real to HMI Analog Output Supply Fan VFD Selected Speed
        [40]   // Zone 2 Real to HMI Parameter TC01 Temperature Zero Offset
        [41]   // Zone 2 Real to HMI Parameter TC02 Temperature Zero Offset
        [42]   // Zone 2 Real to HMI Parameter
        [43]   // Zone 2 Real to HMI Parameter
        [44]   // Zone 2 Real to HMI Parameter PID1 NKp
        [45]   // Zone 2 Real to HMI Parameter PID1 Ki
        [46]   // Zone 2 Real to HMI Parameter PID1 Kd
        [47]   // Zone 2 Real to HMI Parameter PID1 Bias
        [48]   // Zone 2 Real to HMI Parameter PID2 Kp
        [49]   // Zone 2 Real to HMI Parameter PID2 Ki
        [50]   // Zone 2 Real to HMI Parameter PID2 Kd
        [51]   // Zone 2 Real to HMI Parameter PID2 Bias
        [52]   // Zone 2 Real to HMI Parameter Process Control High Limit
        [53]   // Zone 2 Real to HMI Parameter Spare
        [54]   // Zone 2 Real to HMI parameter Process Control Deviation
        [55]   // Zone 2 Real to HMI Parameter LFL Warning Level
        [56]   // Zone 2 Real to HMI Parameter LFL Alarm Level
        [57]   // Zone 2 Real to HMI Parameter Zone Shutdown Temperature
        [58]   // Zone 2 Real to HMI Parameter High Pressure LImit
        [59]   // Zone 2 Real to HMI Temperature Control Fast to Soak Control Deviation
        [60]   // Zone 2 Real to HMI Temperature Control Soak to Fast Control Deviation
        [61]   // Zone 2 Real to HMI Parameter
        [62]   // Zone 2 Real to HMI Parameter
        [63]   // Zone 2 Real to HMI Parameter
        [64]   // Zone 2 Real to HMI Exhaust VFD RPM Setpoint
        [65]   // Zone 2 Real to HMI Recirc VFD RPM Setpoint
        [67]   // Zone 2 Real to HMI Temperature Control Setpoint
        [68]   // Zone 2 Real to HMI Temperature Control manual Control Valve Setpoint
        [69]   // Zone 2 Real to HMI
        [70]   // Zone 2 Real to HMI
        [71]   // Zone 2 Real to HMI
        [72]   // Zone 2 Real to HMI Process Control Temperature
        [73]   // Zone 2 Real to HMI
        [74]   // Zone 2 Real to HMI
        [75]   // Zone 2 Real to HMI
        [76]   // Zone 2 Real to HMI
        [77]   // Zone 2 Real to HMI
        [78]   // Zone 2 Real to HMI
        [79]   // Zone 2 Real to HMI
   p12_recirc_input_max : REAL := 1750.0;
   p12_recirc_input_min : REAL;
   p12_recirc_output_max : REAL := 1750.0;
   p12_recirc_output_min : REAL;
   p12r01 : routine := (comment := 7);   // Zone 2 Main
   p12r02 : routine := (comment := -1073741761);   // Zone 2 Misc Control
        .FAULT.0   // Zone 2 Misc Control
        .WARNING.0   // Zone 2 Misc Control Low Pressure
        .UNACK_FAULT   // Zone 2 Misc Control Unacknowledged Fault Exists
        .UNACK_WARNING   // Zone 2 Misc Control Unacknowledged Warning Exists
   p12r02_fault_exists : BOOL;
   p12r02_not_safe_temp : BOOL := 1;   // Zone 2 Misc Control Zone above Safe Temp
   p12r02_safe_temp : BOOL;   // Zone 2 Misc Control Zone Temperature at Safe Temp
   p12r02_shutdown_temp : BOOL;   // Zone 2 Misc Control Safe Shutdown Temperature
   p12r02_timer_fault : TIMER[4];   // Zone 2 Misc Control Fault Delay
   p12r02_timer_safe_temp : TIMER[2] := ([0].PRE := 30000, [1].PRE := 30000, [1].ACC := 30007, [1].EN := 1, [1].DN := 1);   // Zone 2 Misc Control Chamber SafeTemperature Dwell
   p12r02_timer_warning : TIMER[4] := ([0].PRE := 1500);   // Zone 2 Misc Control Warning Delay
   p12r02_unack_fault : BOOL;   // Zone 2 Misc Control Unacknowledged Fault Exists
   p12r02_unack_warning : BOOL;   // Zone 2 Misc Control Unacknowledged Warning Exists
   p12r02_warning_exists : BOOL := 1;
   p12r03 : routine := (comment := -1073741761);   // Zone 2 Input
        .UNACK_FAULT   // Zone 2 Input Unacknowledged Fault Exists
        .UNACK_WARNING   // Zone 2 Input Unacknowledged Warning Exists
   p12r03_hz : SYS_SCP := (Input := 901.0, Input_Max := 1750.0, Output_Max := 60.0, Output := 30.891432);   // Zone 2 Analog Inputs SCP Hz
   p12r03_timer_fault : TIMER[4];   // Zone 2 Input Fault Delay
   p12r03_timer_warning : TIMER[4];   // Zone 2 Input Warning Delay
   p12r04 : routine := (comment := -1073741761);   // Zone 2 Output
        .UNACK_FAULT   // Zone 2 Analog Output Unacknowledged Fault Exists
        .UNACK_WARNING   // Zone 2 Analog Output Unacknowledged Warning Exists
   p12r04_timer_fault : TIMER[4];   // Zone 2 Output Fault Delay
   p12r04_timer_warning : TIMER[4];   // Zone 2 Output Warning Delay
   p12r05 : routine := (comment := -1073741761);   // Zone 2 Dint to HMI
        .UNACK_FAULT   // Zone 2 Dint to HMI Unacknowledged Fault Exists
        .UNACK_WARNING   // Zone 2 Dint to HMI Unacknowledged Warning Exists
   p12r05_exh_status : DINT := 2;
   p12r05_recirc_status : DINT := 2;
   p12r05_Temp_ctl_status : DINT := 2;
   p12r05_timer_fault : TIMER[4];   // Zone 2 Dint to HMI Fault Delay
   p12r05_timer_warning : TIMER[4];   // Zone 2 Dint to HMI Warning Delay
   p12r06 : routine := (comment := -1073741572);   // Zone 2 Real to HMI
        .UNACK_FAULT   // Zone 2 Real to HMI Unacknowledged Fault Exists
        .UNACK_WARNING   // Zone 2 Real to HMI Unacknowledged Warning Exists
   p12r06_timer_fault : TIMER[4];   // Zone 2 Real to HMI Fault Delay
   p12r06_timer_warning : TIMER[4];   // Zone 2 Real to HMI Warning Delay
   p12r07 : routine := (comment := -1073741761);   // Zone 2 Alarms
        .UNACK_FAULT   // Zone 2 Alarms Unacknowledged Fault Exists
        .UNACK_WARNING   // Zone 2 Alarms Unacknowledged Warning Exists
   p12r07_timer_fault : TIMER[4];   // Zone 2 Alarms Fault Delay
   p12r07_timer_warning : TIMER[4];   // Zone 2 Alarms Warning Delay
   p12r08 : routine := (comment := -1073741761);   // Zone 2 Warnings
        .UNACK_FAULT   // Zone 2 Warnings Unacknowledged Fault Exists
        .UNACK_WARNING   // Zone 2 Warnings Unacknowledged Warning Exists
   p12r08_timer_fault : TIMER[4];   // Zone 2 Warnings Fault Delay
   p12r08_timer_warning : TIMER[4];   // Zone 2 Warnings Warning Delay
   p12r09 : routine := (comment := -1073741761);   // Zone 2 Modes
        .FAULT.0   // Zone 2 Modes
        .UNACK_FAULT   // Zone 2 Modes Unacknowledged Fault Exists
        .UNACK_WARNING   // Zone 2 Modes Unacknowledged Warning Exists
   p12r09_timer_fault : TIMER[4];   // Zone 2 Modes Fault Delay
   p12r09_timer_warning : TIMER[8];   // Zone 2 Modes Warning Delay
   p12r10 : routine := (comment := -1073741761);   // Zone 2
        .UNACK_FAULT   // Zone 2 Unacknowledged Fault Exists
        .UNACK_WARNING   // Zone 2 Unacknowledged Warning Exists
   p12r10_timer_fault : TIMER[4];   // Zone 2 Fault Delay
   p12r10_timer_warning : TIMER[4];   // Zone 2 Warning Delay
   p12r15_mtr_roll_speed_offset : REAL;   // Impreg Metering Roll VFD Speed Offset
   p12r16_pid_temp_cv : DINT := 27;   // Zone 2 Temperature Control Control Valve
   p12r16_temp_ok : BOOL := 1;   // Zone 2 Temperature Control Temperature OK
   p12r20 : routine := (comment := -1073741761);   // Zone 2 Temp Sequence
        .FAULT.0   // Zone 2
        .FAULT.1   // Zone 2
        .FAULT.2   // Zone 2
        .FAULT.3   // Zone 2
        .WARNING.0   // Zone 2
        .UNACK_FAULT   // Zone 2 Temp Sequence Unacknowledged Fault Exists
        .UNACK_WARNING   // Zone 2 Unacknowledged Warning Exists
   p12r20_safeties_ok : BOOL := 1;   // Zone 2 Temperature Control Burner Safeties OK this Lightoff
   p12r20_state : DINT := 1025;   // Zone 2 Temperature Control State
        .0   // Zone 2 Temperature Control State 0 One-Step per Scan
        .1   // Zone 2 Temperature Control State 1 Off
        .2   // Zone 2 Temperature Control State 2 Idle
        .3   // Zone 2 Temperature Control State 3 Start Recirculation Fan
        .4   // Zone 2 Temperature Control State 4 Start Exhaust Fan
        .5   // Zone 2 Temperature Control State 5 Wait for Safeties
        .6   // Zone 2 Temperature Control State 6 Safeties Made
        .7   // Zone 2 Temperature Control State 7 Purge
        .8   // Zone 2 Temperature Control State 8 Burner Lit
        .9   // Zone 2 Temperature Control State 9 Heat to Setpoint
        .10   // Zone 2 Temperature Control State 10 Control to Setpoint
        .11   // Zone 2 Temperature Control State 11 Cooldown
        .12   // Zone 2 Temperature Control State 12 Cooldown Fans
        .13   // Zone 2 Temperature Control State 13 Complete
        .31   // Zone 2 Temperature Control State 31 Manual
   p12r20_status : DINT := 10;   // Zone 2 Temperature Control Sequence Status
   p12r20_timer_fault : TIMER[4];   // Zone 2 Temp Sequence Fault Delay
   p12r20_timer_state_11 : TIMER := (PRE := 5000);   // Zone 2 Temp Sequence State 11 Dwell
   p12r20_timer_state_3 : TIMER := (PRE := 1000, ACC := 1022, EN := 1, DN := 1);   // Zone 2 Temperature Control State 3 Dwell
   p12r20_timer_state_4 : TIMER := (PRE := 1000, ACC := 1025, EN := 1, DN := 1);   // Zone 2 Temp Sequence State 4 Dwell
   p12r20_timer_state_7 : TIMER := (PRE := 2000, ACC := 2020, EN := 1, DN := 1);   // Zone 2 Temp Sequence State 7 Dwell
   p12r20_timer_warning : TIMER[4];   // Zone 2 Temp Sequence Warning Delay
   p12r30 : routine := (comment := -1073741697, oneshot := 4, warning := 192, warning_ack := 192);   // Zone 2 Temperature Control
        .FAULT.0   // Zone 2 Temperature Control Process Control Software High Limit
        .FAULT.1   // Zone 2 Temperature Control Process Control Hardware High Limit
        .FAULT.2   // Zone 2 Temperature Control Process Control Thermocouple Failure
        .FAULT.3   // Zone 2 Temperature Control Process Control Temperature Spare
        .FAULT.4   // Zone 2 Temperature Control Lower Flash Limit High High Limit Exceeded
        .FAULT.5   // Zone 2 Temperature Control Flame Failure
        .FAULT.6   // Zone 2 Temperature Control Burner Safeties Failure
        .FAULT.7   // Zone 2 Temperature Control Recirculation Fan Speed Fault
        .FAULT.8   // Zone 2 Temperature Control Exhaust Fan Speed Fault
        .FAULT.9   // Zone 2 Temperature Control Access Door Open
        .FAULT.10   // Zone 2 Temperature Control Spare
        .FAULT.11   // Zone 2 Temperature Control
        .FAULT.12   // Zone 2 Temperature Control Spare
        .FAULT.13   // Zone 2 Temperature Control
        .FAULT.14   // Zone 2 Temperature Control
        .WARNING.0   // Zone 2 Temperature Control Control Temperature Deviation
        .WARNING.1   // Zone 2 Temperature Control Process Control Thermocouple 1 Failure
        .WARNING.2   // Zone 2 Temperature Control Process Control Thermocouple 2 Failure
        .WARNING.3   // Zone 2 Temperature Control Control Valve in Manual
        .WARNING.4   // Zone 2 Temperature Control LFL High Limit
        .WARNING.5   // Zone 2 Temperature Control Zone Off
        .WARNING.6   // Zone 2 Temperature Control Fresh Air Filter Dirty
        .WARNING.7   // Zone 2 Temperature Control Combustion Air Filter Dirty
        .WARNING.8   // Zone 2 Temperature Control Recirculation Air Filter Dirty
        .UNACK_FAULT   // Zone 2 Temperature Control Unacknowledged Fault Exists
        .UNACK_WARNING   // Zone 2 Temperature Control Unacknowledged Warning Exists
   p12r30_cv_man_sp : REAL := 60.0;   // Zone 2 Temperature Control Manual Heat Control Valve Setpoint
   p12r30_pb_auto : BOOL;   // Zone 2 Temperature Control PB: Zone Control Auto
   p12r30_pb_manual : BOOL;   // Zone 2 Temperature Control PB: Zone Control Manual
   p12r30_pb_zone_off : BOOL;   // Zone 2 Temperature Control PB: Stop Zone Heat Control
   p12r30_pb_zone_on : BOOL;   // Zone 2 Temperature Control PB: Start Zone Heat Control
   p12r30_permissive_run : BOOL := 1;   // Zone 2 Temperature Control Run Permissive
   p12r30_pid_temp : PID := (CTL := -2144304512, EN := 1, NOBC := 1, NOZC := 1, INI := 1, DVPA := 1, PVHA := 1, SP := 200.0, KP := 20.0, KI := 0.5, BIAS := 15.0, MAXS := 1000.0, SO := 27.039719, MAXO := 100.0, UPD := 0.01, PV := 199.5, ERR := 0.5, OUT := 27.039719, MAXI := 10000.0, MAXCV := 100.0, MAXTIE := 4095.0, DATA[0] := 11.03972, DATA[1] := -319.2, DATA[2] := 199.5, DATA[3] := 0.5, DATA[4] := 200.0, DATA[5] := 0.1, DATA[6] := 0.1, DATA[7] := 0.16, DATA[8] := 20.0, DATA[9] := 0.5, DATA[11] := 20.0, DATA[12] := 0.5, DATA[15] := 1.0, DATA[16] := 0.024420025);   // Zone 2 Temperature Control PID
   p12r30_pid_temp_pv : REAL := 1994.0001;   // Zone 2 Temperature Control PID Temp Process Variable
   p12r30_pid_temp_sp : REAL := 200.0;   // Zone 2 Temperature Control PID Temperature Control Setpoint
   p12r30_pid_temp_sp_error : REAL := 0.59999084;   // Zone 2 Temperature Control Setpoint/Process Variable Error (ABS)
   p12r30_pid_temp_sp_last : REAL := 200.0;   // Zone 2 Temperature Control Setpoint Last Scan
   p12r30_request_deviation_warning : BOOL := 1;   // Zone 2 Temperature Control Request Setpoint Deviation Warning
   p12r30_request_heat : BOOL := 1;   // Zone 2 Temperature Control Request Heat
   p12r30_request_heat_last : BOOL := 1;   // Zone 2 Temperature Control Request Heat Last Scan
   p12r30_request_manual : BOOL;   // Zone 2 Temperature Control Request Manual Control
   p12r30_request_PID_shot : BOOL;
   p12r30_request_soak_control : BOOL := 1;   // Zone 2 Temperature Control Request Soak Control
   p12r30_temp_deviation_setpoint : DINT := 5;
   p12r30_timer_fault : TIMER[16] := ([0].PRE := 5000, [2].PRE := 1000, [4].PRE := 1000, [10].PRE := 5000, [11].PRE := 5000, [12].PRE := 5000);   // Zone 2 Temperature Control Fault Delay
   p12r30_timer_warning : TIMER[12] := ([0].PRE := 10000, [1].PRE := 1000, [2].PRE := 1000, [3].PRE := 90000, [4].PRE := 1000, [6].PRE := 1000, [6].ACC := 1029, [6].EN := 1, [6].DN := 1, [7].PRE := 1000, [7].ACC := 1029, [7].EN := 1, [7].DN := 1, [8].PRE := 1000);   // Zone 2 Temperature Control Warning Delay
   p12r30_vfds_ok : BOOL := 1;
   p12r30_vfds_ready : BOOL := 1;   // Zone 2 Temperature Control VFDs On
   p12r31 : routine := (comment := -1073741697);   // Zone 2 Exhaust VFD
        .FAULT.0   // Zone 2 Exhaust VFD Drive Fault
        .FAULT.1   // Zone 2 Exhaust VFD Motor Thermistor Not OK
        .FAULT.2   // Zone 2 Exhaust VFD Not Ready
        .FAULT.3   // Zone 2 Exhaust VFD
        .WARNING.0   // Zone 2 Exhaust VFD VFD Stopped While Chamber is Too Hot
        .WARNING.1   // Zone 2 Exhaust VFD Fan Flow Failure
        .WARNING.2   // Zone 2 Exhaust VFD VFD Warning
        .UNACK_FAULT   // Zone 2 Exhaust VFD Unacknowledged Fault Exists
        .UNACK_WARNING   // Zone 2 Exhaust VFD Unacknowledged Warning Exists
   p12r31_pb_start : BOOL;   // Zone 2 Exhaust VFD PB: Start
   p12r31_pb_stop : BOOL;   // Zone 2 Exhaust VFD PB: Stop
   p12r31_request_auto_run : BOOL := 1;   // Zone 2 Exhaust Fan Run Request
   p12r31_request_auto_stop : BOOL := 1;   // Zone 2 Exhaust VFD Request Auto Stop
   p12r31_run_permissive : BOOL := 1;   // Zone 2 Exhaust VFD Run Permissive
   p12r31_timer_fault : TIMER[5] := ([1].PRE := 500);   // Zone 2 Exhaust VFD Fault Timer
   p12r31_timer_warning : TIMER[5] := ([0].PRE := 10000, [1].PRE := 20000, [2].PRE := 500);   // Zone 2 Exhaust VFD Waringing Timer
   p12r31_vfd_stopped : BOOL;   // Zone 2 Exhaust VFD VFD Stopped
   p12r32 : routine := (comment := -536870849);   // Zone 2 Recirc VFD
        .FAULT.0   // Zone 2 Recirc VFD Drive Fault
        .FAULT.1   // Zone 2 Recirc VFD Motor Thermistor Not OK
        .FAULT.2   // Zone 2 Recirc VFD Not Ready
        .FAULT.3   // Zone 2 Supply VFD
        .WARNING.0   // Zone 2 Recirc VFD VFD Stopped While Chamber is Too Hot
        .WARNING.1   // Zone 2 Recirc VFD Fan Flow Failure
        .WARNING.2   // Zone 2 Recirc VFD VFD Warning
        .UNACK_FAULT   // Zone 2 Recirc VFD Unacknowledged Fault Exists
        .UNACK_WARNING   // Zone 2 Recirc VFD Unacknowledged Warning Exists
   p12r32_fan_pb_stopped : BOOL;   // Zone 2 Recirc VFD Fan Stopped Manually - Prevent Auto Start during Cooldown
   p12r32_pb_start : BOOL;   // Zone 2 Recirc VFD PB: Start
   p12r32_pb_stop : BOOL;   // Zone 2 Recirc VFD PB: Stop
   p12r32_request_auto_run : BOOL := 1;   // Zone 2 Recirc Fan Run Request
   p12r32_request_auto_stop : BOOL := 1;   // Zone 2 Recirc VFD Request Auto Stop
   p12r32_run_permissive : BOOL := 1;   // Zone 2 Recirc VFD Run Permissive
   p12r32_timer_fault : TIMER[5] := ([1].PRE := 500);   // Zone 2 Recirc VFD Fault Timer
   p12r32_timer_warning : TIMER[5] := ([0].PRE := 10000, [1].PRE := 20000, [2].PRE := 20000);   // Zone 2 Supply VFD Warning Timer
   p12r32_vfd_stopped : BOOL;   // Zone 2 Recirc VFD VFD Stopped
   p13_ai_exhaust_amps : REAL := 0.8;   // Zone 3 Analog Input Exhaust Fan Amps
   p13_ai_exhaust_hz : REAL := 30.891432;   // Zone 3 Analog Input Exhaust Fan HZ
   p13_ai_exhaust_hz_max : REAL := 60.0;   // Zone 3 Analog Input Exhaust Fan Max HZ
   p13_ai_exhaust_pct : REAL;   // Zone 3 Analog Input Exhaust Fan PCT
   p13_ai_exhaust_rpm : REAL := 901.0;   // Zone 3 Analog Input Exhaust Fan RPM
   p13_ai_recirc_amps : REAL := 7.9;   // Zone 3 Analog Input Recirc Fan Amps
   p13_ai_recirc_hz : REAL := 44.605717;   // Zone 3 Analog Input Supply Fan HZ
   p13_ai_recirc_hz_max : REAL := 60.0;   // Zone 3 Analog Input Supply Fan max HZ
   p13_ai_recirc_pct : REAL;   // Zone 3 Analog Input Recirc Fan PCT
   p13_ai_recirc_rpm : REAL := 1301.0;   // Zone 3 Analog Input Recirc Fan RPM
   p13_ai_tc01 : REAL := 66.3;   // Zone 3 Analog Input Control Thermocouple 1
   p13_ai_tc02 : REAL := 65.6;   // Zone 3 Analog Input Control Thermocouple 2
   p13_ao_cv : REAL := 100.0;   // Zone 3 Analog Output Control Valve
   p13_ao_exhaust_selected_speed : REAL := 900.0;   // Zone 3 Analog Output Exhaust Fan VFD Selected Speed
   p13_ao_recirc_selected_speed : REAL := 1300.0;   // Zone 3 Analog Output Recirc Fan VFD Selected Speed
   p13_di_door_open : BOOL;   // Zone 3 Digital Input Access Door Open
   p13_di_exh : acs800_di_normal := (running_fwd := 1, ready := 1, ctrl_from_net := 1, ref_from_net := 1, at_reference := 1);   // Zone 3 Digital Inputs Exhaust Fan
        .FAULTED   // Zone 3 Digital Inputs Exhaust Fan
   p13_di_exh_fan_mtr_ts : BOOL := 1;   // Zone 3 Digital Input Exhaust Fan Motor Thermostat OK
   p13_di_exh_flow_ok : BOOL := 1;   // Zone 3 Digital Input Exhaust Flow OK
   p13_di_filter_clean : BOOL := 1;   // Zone 3 Digital Input Filter Dirty
   p13_di_recirc : acs800_di_normal := (running_fwd := 1, ready := 1, ctrl_from_net := 1, ref_from_net := 1, at_reference := 1);   // Zone 3 Digital Inputs Recirc Fan
   p13_di_recirc_fan_mtr_ts : BOOL := 1;   // Zone 3 Digital Input Recirc Fan Motor Thermostat OK
   p13_di_recirc_flow_ok : BOOL := 1;   // Zone 3 Digital Input Recirc Flow OK
   p13_di_tc01_bo : BOOL;   // Zone 3 Digital Input Control Thermocouple 1 Failure
   p13_di_tc02_bo : BOOL;   // Zone 3 Digital Input Control Thermocouple 2 Failure
   p13_dint_to_hmi : DINT[16] := ([4] := 590163, [5] := 16845924, [6] := 62708, [8] := 5, [9] := 2, [10] := 2, [11] := 2);   // Zone 3 Temperature Control VFDs On
        [0]   // Zone 3 Dint to HMI Alarms
        [0].0   // Zone 3 Dint to HMI Alarms A00:
        [0].1   // Zone 3 Dint to HMI Alarms A01:
        [0].2   // Zone 3 Dint to HMI Alarms A02: Process Control Thermocouple Failure
        [0].3   // Zone 3 Dint to HMI Alarms A03:
        [0].4   // Zone 3 Dint to HMI Alarms A04:
        [0].5   // Zone 3 Dint to HMI Alarms A05:
        [0].6   // Zone 3 Dint to HMI Alarms A06:
        [0].7   // Zone 3 Dint to HMI Alarms A07:
        [0].8   // Zone 3 Dint to HMI Alarms A08:
        [0].9   // Zone 3 Dint to HMI Alarms A09: Access Door Open
        [0].10   // Zone 3 Dint to HMI Alarms A10:
        [0].11   // Zone 3 Dint to HMI Alarms A11:
        [0].12   // Zone 3 Dint to HMI Alarms A12:
        [0].13   // Zone 3 Dint to HMI Alarms A13:
        [0].14   // Zone 3 Dint to HMI Alarms A14:
        [0].15   // Zone 3 Dint to HMI Alarms A15:
        [0].16   // Zone 3 Dint to HMI Alarms A16: Exhaust Fan Drive Fault
        [0].17   // Zone 3 Dint to HMI Alarms A17: Exhaust Fan Motor Thermistor Not OK
        [0].18   // Zone 3 Dint to HMI Alarms A18: Exhaust Fan VFD Not Ready
        [0].19   // Zone 3 Dint to HMI Alarms A19:
        [0].20   // Zone 3 Dint to HMI Alarms A20: Recirculation Fan Drive Fault
        [0].21   // Zone 3 Dint to HMI Alarms A21: Recirculation Fan Motor Thermistor Not OK
        [0].22   // Zone 3 Dint to HMI Alarms A22: Recirculation Fan VFD Not Ready
        [0].23   // Zone 3 Dint to HMI Alarms A23:
        [0].24   // Zone 3 Dint to HMI Alarms A24:
        [0].25   // Zone 3 Dint to HMI Alarms A25:
        [0].26   // Zone 3 Dint to HMI Alarms A26:
        [0].27   // Zone 3 Dint to HMI Alarms A27:
        [0].28   // Zone 3 Dint to HMI Alarms A28:
        [0].29   // Zone 3 Dint to HMI Alarms A29:
        [0].30   // Zone 3 Dint to HMI Alarms A30:
        [0].31   // Zone 3 Dint to HMI Alarms A31:
        [1]   // Zone 3 Dint to HMI Alarms
        [1].0   // Zone 3 Dint to HMI Alarms
        [1].1   // Zone 3 Dint to HMI Alarms
        [1].2   // Zone 3 Dint to HMI Alarms
        [1].3   // Zone 3 Dint to HMI Alarms
        [1].4   // Zone 3 Dint to HMI Alarms
        [1].5   // Zone 3 Dint to HMI Alarms
        [1].6   // Zone 3 Dint to HMI Alarms
        [1].7   // Zone 3 Dint to HMI Alarms
        [1].8   // Zone 3 Dint to HMI Alarms
        [1].9   // Zone 3 Dint to HMI Alarms
        [1].10   // Zone 3 Dint to HMI Alarms
        [1].11   // Zone 3 Dint to HMI Alarms
        [1].12   // Zone 3 Dint to HMI Alarms
        [1].13   // Zone 3 Dint to HMI Alarms
        [1].14   // Zone 3 Dint to HMI Alarms
        [1].15   // Zone 3 Dint to HMI Alarms
        [1].16   // Zone 3 Dint to HMI Alarms
        [1].17   // Zone 3 Dint to HMI Alarms
        [1].18   // Zone 3 Dint to HMI Alarms
        [1].19   // Zone 3 Dint to HMI Alarms
        [1].20   // Zone 3 Dint to HMI Alarms
        [1].21   // Zone 3 Dint to HMI Alarms
        [1].22   // Zone 3 Dint to HMI Alarms
        [1].23   // Zone 3 Dint to HMI Alarms
        [1].24   // Zone 3 Dint to HMI Alarms
        [1].25   // Zone 3 Dint to HMI Alarms
        [1].26   // Zone 3 Dint to HMI Alarms
        [1].27   // Zone 3 Dint to HMI Alarms
        [1].28   // Zone 3 Dint to HMI Alarms
        [1].29   // Zone 3 Dint to HMI Alarms
        [1].30   // Zone 3 Dint to HMI Alarms
        [1].31   // Zone 3 Dint to HMI Alarms
        [2]   // Zone 3 Dint to HMI Warnings
        [2].0   // Zone 3 Dint to HMI Warnings W00: Control Temperature Deviation
        [2].1   // Zone 3 Dint to HMI Warnings W01: Process Control Thermocouple 1 Failure
        [2].2   // Zone 3 Dint to HMI Warnings W02: Process Control Thermocouple 2 Failure
        [2].3   // Zone 3 Dint to HMI Warnings W03: Control Valve in Manual
        [2].4   // Zone 3 Dint to HMI Warnings W04: LFL High Limit
        [2].5   // Zone 3 Dint to HMI Warnings W05:
        [2].6   // Zone 3 Dint to HMI Warnings W06: Fresh Air Filter Dirty
        [2].7   // Zone 3 Dint to HMI Warnings W07: Combustion Air Filter Dirty
        [2].8   // Zone 3 Dint to HMI Warnings W08: Recirculation Air Filter Dirty
        [2].9   // Zone 3 Dint to HMI Warnings W09:
        [2].10   // Zone 3 Dint to HMI Warnings W10:
        [2].11   // Zone 3 Dint to HMI Warnings W11:
        [2].12   // Zone 3 Dint to HMI Warnings W12:
        [2].13   // Zone 3 Dint to HMI Warnings W13:
        [2].14   // Zone 3 Dint to HMI Warnings W14:
        [2].15   // Zone 3 Dint to HMI Warnings W15: Low Pressure
        [2].16   // Zone 3 Dint to HMI Warnings W16: Exhaust Fan Stopped While Zone is Too Hot
        [2].17   // Zone 3 Dint to HMI Warnings W17:
        [2].18   // Zone 3 Dint to HMI Warnings W18:
        [2].19   // Zone 3 Dint to HMI Warnings W19:
        [2].20   // Zone 3 Dint to HMI Warnings W20: Recirculation Fan Stopped While Zone is Too Hot
        [2].21   // Zone 3 Dint to HMI Warnings W21: Recirculation Fan Flow Failure
        [2].22   // Zone 3 Dint to HMI Warnings W22: Recirculation Fan Pressure Failure
        [2].23   // Zone 3 Dint to HMI Warnings W23:
        [2].24   // Zone 3 Dint to HMI Warnings W24:
        [2].25   // Zone 3 Dint to HMI Warnings W25:
        [2].26   // Zone 3 Dint to HMI Warnings W26:
        [2].27   // Zone 3 Dint to HMI Warnings W27:
        [2].28   // Zone 3 Dint to HMI Warnings W28:
        [2].29   // Zone 3 Dint to HMI Warnings W29:
        [2].30   // Zone 3 Dint to HMI Warnings W30:
        [2].31   // Zone 3 Dint to HMI Warnings W31:
        [3]   // Zone 3 Dint to HMI Warnings
        [3].0   // Zone 3 Dint to HMI Alarms
        [3].1   // Zone 3 Dint to HMI Alarms
        [3].2   // Zone 3 Dint to HMI Alarms
        [3].3   // Zone 3 Dint to HMI Alarms
        [3].4   // Zone 3 Dint to HMI Alarms
        [3].5   // Zone 3 Dint to HMI Alarms
        [3].6   // Zone 3 Dint to HMI Alarms
        [3].7   // Zone 3 Dint to HMI Alarms
        [3].8   // Zone 3 Dint to HMI Alarms
        [3].9   // Zone 3 Dint to HMI Alarms
        [3].10   // Zone 3 Dint to HMI Alarms
        [3].11   // Zone 3 Dint to HMI Alarms
        [3].12   // Zone 3 Dint to HMI Alarms
        [3].13   // Zone 3 Dint to HMI Alarms
        [3].14   // Zone 3 Dint to HMI Alarms
        [3].15   // Zone 3 Dint to HMI Alarms
        [3].16   // Zone 3 Dint to HMI Alarms
        [3].17   // Zone 3 Dint to HMI Alarms
        [3].18   // Zone 3 Dint to HMI Alarms
        [3].19   // Zone 3 Dint to HMI Alarms
        [3].20   // Zone 3 Dint to HMI Alarms
        [3].21   // Zone 3 Dint to HMI Alarms
        [3].22   // Zone 3 Dint to HMI Alarms
        [3].23   // Zone 3 Dint to HMI Alarms
        [3].24   // Zone 3 Dint to HMI Alarms
        [3].25   // Zone 3 Dint to HMI Alarms
        [3].26   // Zone 3 Dint to HMI Alarms
        [3].27   // Zone 3 Dint to HMI Alarms
        [3].28   // Zone 3 Dint to HMI Alarms
        [3].29   // Zone 3 Dint to HMI Alarms
        [3].30   // Zone 3 Dint to HMI Alarms
        [3].31   // Zone 3 Dint to HMI Alarms
        [4]   // Zone 3 Dint to HMI Process Indicators
        [4].0   // Zone 3 Dint to HMI PI: Zone Fault
        [4].1   // Zone 3 Dint to HMI PI: VFDs On\Ready
        [4].2   // Zone 3 Dint to HMI PI:
        [4].3   // Zone 3 Dint to HMI PI:
        [4].4   // Zone 3 Dint to HMI Exhaust VFD PI: Request Auto Run
        [4].5   // Zone 3 Dint to HMI Exhaust VFD PI: VFD Stopped
        [4].6   // Zone 3 Dint to HMI Exhaust VFD PI: Request Auto Stop
        [4].7   // Zone 3 Dint to HMI Exhaust VFD PI:
        [4].8   // Zone 3 Dint to HMI Recirc VFD PI: Request Auto Run
        [4].9   // Zone 3 Dint to HMI Recirc VFD PI: VFD Stopped
        [4].10   // Zone 3 Dint to HMI Recirc VFD PI: Request Auto Stop
        [4].11   // Zone 3 Dint to HMI Supply VFD PI:
        [4].12   // Zone 3 Dint to HMI PI:
        [4].13   // Zone 3 Dint to HMI PI:
        [4].14   // Zone 3 Dint to HMI PI:
        [4].15   // Zone 3 Dint to HMI PI:
        [4].16   // Zone 3 Dint to HMI Temperature Control PI: Request Heat
        [4].17   // Zone 3 Dint to HMI Temperature Control PI: Off
        [4].18   // Zone 3 Dint to HMI Temperature Control PI: Request Manual Control
        [4].19   // Zone 3 Dint to HMI Temperature Control PI: Request Auto Control
        [4].20   // Zone 3 Dint to HMI PI:
        [4].21   // Zone 3 Dint to HMI PI:
        [4].22   // Zone 3 Dint to HMI PI:
        [4].23   // Zone 3 Dint to HMI PI:
        [4].24   // Zone 3 Dint to HMI PI:
        [4].25   // Zone 3 Dint to HMI PI:
        [4].26   // Zone 3 Dint to HMI PI:
        [4].27   // Zone 3 Dint to HMI PI:
        [4].28   // Zone 3 Dint to HMI PI:
        [4].29   // Zone 3 Dint to HMI PI:
        [4].30   // Zone 3 Dint to HMI PI:
        [4].31   // Zone 3 Dint to HMI PI:
        [5]   // Zone 3 Dint to HMI Process Indicators
        [5].4   // Zone 3 Dint to HMI PI: Digital Input Access Door Open
        [5].5   // Zone 3 Dint to HMI PI: Digital Input Exhaust Fan Motor Thermostat OK
        [5].6   // Zone 3 Dint to HMI PI: Digital Input Exhaust Flow OK
        [5].10   // Zone 3 Dint to HMI PI: Digital Input Recirc Fan Motor Thermostat OK
        [5].11   // Zone 3 Dint to HMI PI: Digital Input Recirc Flow OK
        [5].14   // Zone 3 Dint to HMI PI: Digital Input Control Thermocouple 1 Failure
        [5].15   // Zone 3 Dint to HMI PI: Digital Input Control Thermocouple 2 Failure
        [6]   // Zone 3 Dint to HMI
        [6].0   // Zone 3 Dint to HMI Exhaust VFD Faulted
        [6].1   // Zone 3 Dint to HMI Exhaust VFD Warning
        [6].2   // Zone 3 Dint to HMI Exhaust VFD Running Forward
        [6].3   // Zone 3 Dint to HMI Exhaust VFD Running Reverse
        [6].4   // Zone 3 Dint to HMI Exhaust VFD Ready
        [6].5   // Zone 3 Dint to HMI Exhaust VFD Control from Net
        [6].6   // Zone 3 Dint to HMI Exhaust VFD Reference from Net
        [6].7   // Zone 3 Dint to HMI Exhaust VFD At Reference
        [6].8   // Zone 3 Dint to HMI Recirc VFD Faulted
        [6].9   // Zone 3 Dint to HMI Recirc VFD Warning
        [6].10   // Zone 3 Dint to HMI Recirc VFD Running Forward
        [6].11   // Zone 3 Dint to HMI Recirc VFD Running Reverse
        [6].12   // Zone 3 Dint to HMI Recirc VFD Ready
        [6].13   // Zone 3 Dint to HMI Recirc VFD Control from Net
        [6].14   // Zone 3 Dint to HMI Recirc VFD Reference from Net
        [6].15   // Zone 3 Dint to HMI Recirc VFD At Reference
        [6].16   // Zone 3 Dint to HMI Temperature Control PI: Request Heat
        [6].17   // Zone 3 Dint to HMI Temperature Control PI: Off
        [6].18   // Zone 3 Dint to HMI Temperature Control PI: Request Manual Control
        [6].19   // Zone 3 Dint to HMI Temperature Control PI:
        [6].20   // Zone 3 Dint to HMI PI:
        [6].21   // Zone 3 Dint to HMI PI:
        [6].22   // Zone 3 Dint to HMI PI:
        [6].23   // Zone 3 Dint to HMI PI:
        [6].24   // Zone 3 Dint to HMI PI:
        [6].25   // Zone 3 Dint to HMI PI:
        [6].26   // Zone 3 Dint to HMI PI:
        [6].27   // Zone 3 Dint to HMI PI:
        [6].28   // Zone 3 Dint to HMI PI:
        [6].29   // Zone 3 Dint to HMI PI:
        [6].30   // Zone 3 Dint to HMI PI:
        [6].31   // Zone 3 Dint to HMI PI:
        [7]   // Zone 3 Dint to HMI
        [8]   // Zone 3 Dint to HMI Temperature Control Status - State
        [9]   // Zone 3 Dint to HMI Temperature Control Status (Ready/Fault etc)
        [10]   // Zone 3 Dint to HMI Exhaust VFD Status
        [11]   // Zone 3 Dint to HMI Recirc VFD Status
        [12]   // Zone 3 Dint to HMI
        [13]   // Zone 3 Dint to HMI
        [14]   // Zone 3 Dint to HMI
        [15]   // Zone 3 Dint to HMI
   p13_do_exh : acs800_do_normal := (forward := 1);   // Zone 3 Digital Output Exhaust Fan
   p13_do_recirc : acs800_do_normal := (forward := 1);   // Zone 3 Digital Outputs Supply Fan
   p13_exhaust_input_max : REAL := 2000.0;
   p13_exhaust_input_min : REAL;
   p13_exhaust_output_max : REAL := 2000.0;
   p13_exhaust_output_min : REAL;
   p13_hc_input_max : REAL := 100.0;
   p13_hc_input_min : REAL;
   p13_hc_output_max : REAL := 30840.0;
   p13_hc_output_min : REAL;
   p13_param_fast_to_soak : REAL := 5.0;   // Zone 3 Parameter Fast to Soak Control
   p13_param_lfl_hhl : REAL := 40.0;   // Zone 3 Parameter High High Lower Flash Limit
   p13_param_lfl_hl : REAL := 25.0;   // Zone 3 Parameter High LFL Limit
   p13_param_pid1_ff : REAL;   // Zone 3 Parameter Fast PID Bias
   p13_param_pid1_kd : REAL;   // Zone 3 Parameter Fast PID Derivative Gain
   p13_param_pid1_ki : REAL := 0.1;   // Zone 3 Parameter Fast PID Integral Gain
   p13_param_pid1_kp : REAL := 10.0;   // Zone 3 Parameter Fast PID Proportional Gain
   p13_param_pid2_ff : REAL;   // Zone 3 Parameter Auto PID Bias
   p13_param_pid2_kd : REAL;   // Zone 3 Parameter Auto PID Derivative Gain
   p13_param_pid2_ki : REAL := 1.0;   // Zone 3 Parameter Auto PID Integral Gain
   p13_param_pid2_kp : REAL := 10.0;   // Zone 3 Parameter Auto PID Proportional Gain
   p13_param_shutdown_temp : REAL := 125.0;   // Zone 3 Parameter Zone Shutdown Temperature
   p13_param_soak_to_fast : REAL := 15.0;   // Zone 3 Parameter Soak to Fast Control
   p13_param_tc01_dev : REAL := 50.0;   // Zone 3 Parameter Oven Temperature Deviation from Setpoint
   p13_param_tc01_hl : REAL := 400.0;   // Zone 3 Parameter Process Air High Limit
   p13_param_tc01z : REAL;   // Zone 3 Parameter Process Temperature Zero Offset
   p13_param_tc02z : REAL;   // Zone 3 Parameter SupplyTemperature Zero Offset
   p13_param_zone_pressure : REAL;   // Zone 3 Parameter High Pressure LImit
   p13_real_to_hmi : REAL[112] := ([0] := 65.8, [1] := 65.8, [2] := 65.8, [8] := 30.891432, [9] := 0.8, [10] := 901.0, [12] := 44.605717, [13] := 7.9, [14] := 1301.0, [24] := 100.0, [28] := 900.0, [30] := 1300.0, [44] := 10.0, [45] := 0.1, [48] := 10.0, [49] := 1.0, [52] := 400.0, [54] := 50.0, [55] := 25.0, [56] := 40.0, [57] := 125.0, [59] := 5.0, [60] := 15.0, [67] := 60.0, [68] := 80.0, [72] := 65.8);   // Zone 3 Real to HMI
        [0]   // Zone 3 Real to HMI Analog Input Zone 3 Process Control Temperature 1
        [1]   // Zone 3 Real to HMI Analog Input Zone 3 Process Control Temperature 2
        [2]   // Zone 3 Real to HMI Analog Input
        [3]   // Zone 3 Real to HMI Analog Input
        [6]   // Zone 3 Real to HMI Analog Input Pressure
        [7]   // Zone 3 Real to HMI Analog Input Lower Flash Limit
        [8]   // Zone 3 Real to HMI Analog Input Exhaust Fan Hz
        [9]   // Zone 3 Real to HMI Analog Input Exhaust Fan Amps
        [10]   // Zone 3 Real to HMI Analog Input Exhaust Fan RPM
        [11]   // Zone 3 Real to HMI Analog Input Exhaust Fan PCT
        [12]   // Zone 3 Real to HMI Analog Input Recirc Fan Hz
        [13]   // Zone 3 Real to HMI Analog Input Recirc Fan Amps
        [14]   // Zone 3 Real to HMI Analog Analog Input Recirc Fan RPM
        [15]   // Zone 3 Real to HMI Analog Analog Input Recirc Fan Pct
        [16]   // Zone 3 Real to HMI Analog Input Spare
        [17]   // Zone 3 Real to HMI Analog Input Spare
        [24]   // Zone 3 Real to HMI Analog Output PID Control Value
        [28]   // Zone 3 Real to HMI Analog Output Exhaust Fan VFD Selected Speed
        [30]   // Zone 3 Real to HMI Analog Output Supply Fan VFD Selected Speed
        [40]   // Zone 3 Real to HMI Parameter TC01 Temperature Zero Offset
        [41]   // Zone 3 Real to HMI Parameter TC02 Temperature Zero Offset
        [42]   // Zone 3 Real to HMI Parameter
        [43]   // Zone 3 Real to HMI Parameter
        [44]   // Zone 3 Real to HMI Parameter PID1 NKp
        [45]   // Zone 3 Real to HMI Parameter PID1 Ki
        [46]   // Zone 3 Real to HMI Parameter PID1 Kd
        [47]   // Zone 3 Real to HMI Parameter PID1 Bias
        [48]   // Zone 3 Real to HMI Parameter PID2 Kp
        [49]   // Zone 3 Real to HMI Parameter PID2 Ki
        [50]   // Zone 3 Real to HMI Parameter PID2 Kd
        [51]   // Zone 3 Real to HMI Parameter PID2 Bias
        [52]   // Zone 3 Real to HMI Parameter Process Control High Limit
        [53]   // Zone 3 Real to HMI Parameter Spare
        [54]   // Zone 3 Real to HMI parameter Process Control Deviation
        [55]   // Zone 3 Real to HMI Parameter LFL Warning Level
        [56]   // Zone 3 Real to HMI Parameter LFL Alarm Level
        [57]   // Zone 3 Real to HMI Parameter Zone Shutdown Temperature
        [58]   // Zone 3 Real to HMI Parameter High Pressure LImit
        [59]   // Zone 3 Real to HMI Temperature Control Fast to Soak Control Deviation
        [60]   // Zone 3 Real to HMI Temperature Control Soak to Fast Control Deviation
        [61]   // Zone 3 Real to HMI Parameter
        [62]   // Zone 3 Real to HMI Parameter
        [63]   // Zone 3 Real to HMI Parameter
        [64]   // Zone 3 Real to HMI Exhaust VFD RPM Setpoint
        [65]   // Zone 3 Real to HMI Recirc VFD RPM Setpoint
        [67]   // Zone 3 Real to HMI Temperature Control Setpoint
        [68]   // Zone 3 Real to HMI Temperature Control manual Control Valve Setpoint
        [69]   // Zone 3 Real to HMI
        [70]   // Zone 3 Real to HMI
        [71]   // Zone 3 Real to HMI
        [72]   // Zone 3 Real to HMI Process Control Temperature
        [73]   // Zone 3 Real to HMI
        [74]   // Zone 3 Real to HMI
        [75]   // Zone 3 Real to HMI
        [76]   // Zone 3 Real to HMI
        [77]   // Zone 3 Real to HMI
        [78]   // Zone 3 Real to HMI
        [79]   // Zone 3 Real to HMI
   p13_recirc_input_max : REAL := 2000.0;
   p13_recirc_input_min : REAL;
   p13_recirc_output_max : REAL := 2000.0;
   p13_recirc_output_min : REAL;
   p13r01 : routine := (comment := 7);   // Zone 3 Main
   p13r02 : routine := (comment := -1073741761);   // Zone 3 Misc Control
        .FAULT.0   // Zone 3 Misc Control
        .UNACK_FAULT   // Zone 3 Misc Control Unacknowledged Fault Exists
        .UNACK_WARNING   // Zone 3 Misc Control Unacknowledged Warning Exists
   p13r02_fault_exists : BOOL;
   p13r02_not_safe_temp : BOOL;   // Zone 3 Misc Control Zone above Safe Temp
   p13r02_safe_temp : BOOL := 1;   // Zone 3 Misc Control Zone Temperature at Safe Temp
   p13r02_shutdown_temp : BOOL := 1;   // Zone 3 Misc Control Safe Shutdown Temperature
   p13r02_timer_fault : TIMER[4];   // Zone 3 Misc Control Fault Delay
   p13r02_timer_safe_temp : TIMER[2] := ([0].PRE := 30000, [0].ACC := 30030, [0].EN := 1, [0].DN := 1, [1].PRE := 30000);   // Zone 3 Misc Control Chamber SafeTemperature Dwell
   p13r02_timer_warning : TIMER[4] := ([0].PRE := 1500);   // Zone 3 Misc Control Warning Delay
   p13r02_unack_fault : BOOL;   // Zone 3 Misc Control Unacknowledged Fault Exists
   p13r02_unack_warning : BOOL;   // Zone 3 Misc Control Unacknowledged Warning Exists
   p13r02_warning_exists : BOOL;
   p13r03 : routine := (comment := -1073741761);   // Zone 3 Input
        .UNACK_FAULT   // Zone 3 Input Unacknowledged Fault Exists
        .UNACK_WARNING   // Zone 3 Input Unacknowledged Warning Exists
   p13r03_hz : SYS_SCP := (Input_Max := 1800.0, Output_Max := 60.0, Output := -3.8146973e-06);   // Zone 3 Analog Inputs SCP Hz
   p13r03_timer_fault : TIMER[4];   // Zone 3 Input Fault Delay
   p13r03_timer_warning : TIMER[4];   // Zone 3 Input Warning Delay
   p13r04 : routine := (comment := -1073741761);   // Zone 3 Output
        .UNACK_FAULT   // Zone 3 Analog Output Unacknowledged Fault Exists
        .UNACK_WARNING   // Zone 3 Analog Output Unacknowledged Warning Exists
   p13r04_timer_fault : TIMER[4];   // Zone 3 Output Fault Delay
   p13r04_timer_warning : TIMER[4];   // Zone 3 Output Warning Delay
   p13r05 : routine := (comment := -1073741761);   // Zone 3 Dint to HMI
        .UNACK_FAULT   // Zone 3 Dint to HMI Unacknowledged Fault Exists
        .UNACK_WARNING   // Zone 3 Dint to HMI Unacknowledged Warning Exists
   p13r05_exh_status : DINT := 2;
   p13r05_recirc_status : DINT := 2;
   p13r05_temp_ctl_status : DINT := 2;
   p13r05_timer_fault : TIMER[4];   // Zone 3 Dint to HMI Fault Delay
   p13r05_timer_warning : TIMER[4];   // Zone 3 Dint to HMI Warning Delay
   p13r06 : routine := (comment := -1073741572);   // Zone 3 Real to HMI
        .UNACK_FAULT   // Zone 3 Real to HMI Unacknowledged Fault Exists
        .UNACK_WARNING   // Zone 3 Real to HMI Unacknowledged Warning Exists
   p13r06_timer_fault : TIMER[4];   // Zone 3 Real to HMI Fault Delay
   p13r06_timer_warning : TIMER[4];   // Zone 3 Real to HMI Warning Delay
   p13r07 : routine := (comment := -1073741761);   // Zone 3 Alarms
        .UNACK_FAULT   // Zone 3 Alarms Unacknowledged Fault Exists
        .UNACK_WARNING   // Zone 3 Alarms Unacknowledged Warning Exists
   p13r07_timer_fault : TIMER[4];   // Zone 3 Alarms Fault Delay
   p13r07_timer_warning : TIMER[4];   // Zone 3 Alarms Warning Delay
   p13r08 : routine := (comment := -1073741761);   // Zone 3 Warnings
        .UNACK_FAULT   // Zone 3 Warnings Unacknowledged Fault Exists
        .UNACK_WARNING   // Zone 3 Warnings Unacknowledged Warning Exists
   p13r08_timer_fault : TIMER[4];   // Zone 3 Warnings Fault Delay
   p13r08_timer_warning : TIMER[4];   // Zone 3 Warnings Warning Delay
   p13r09 : routine := (comment := -1073741761);   // Zone 3 Modes
        .FAULT.0   // Zone 3 Modes
        .UNACK_FAULT   // Zone 3 Modes Unacknowledged Fault Exists
        .UNACK_WARNING   // Zone 3 Modes Unacknowledged Warning Exists
   p13r09_timer_fault : TIMER[4];   // Zone 3 Modes Fault Delay
   p13r09_timer_warning : TIMER[8];   // Zone 3 Modes Warning Delay
   p13r10 : routine := (comment := -1073741761);   // Zone 3
        .UNACK_FAULT   // Zone 3 Unacknowledged Fault Exists
        .UNACK_WARNING   // Zone 3 Unacknowledged Warning Exists
   p13r10_timer_fault : TIMER[4];   // Zone 3 Fault Delay
   p13r10_timer_warning : TIMER[4];   // Zone 3 Warning Delay
   p13r16_pid_temp_cv : DINT := 100;   // Zone 3 Temperature Control Control Valve
   p13r20 : routine := (comment := -1073741761);   // Zone 3 Temp Sequence
        .FAULT.0   // Zone 3
        .FAULT.1   // Zone 3
        .FAULT.2   // Zone 3
        .FAULT.3   // Zone 3
        .WARNING.0   // Zone 3
        .UNACK_FAULT   // Zone 3 Temp Sequence Unacknowledged Fault Exists
        .UNACK_WARNING   // Zone 3 Unacknowledged Warning Exists
   p13r20_state : DINT := 33;   // Zone 3 Temperature Control State
        .0   // Zone 3 Temperature Control State 0 One-Step per Scan
        .1   // Zone 3 Temperature Control State 1 Off
        .2   // Zone 3 Temperature Control State 2 Idle
        .3   // Zone 3 Temperature Control State 3 Start Recirculation Fan
        .4   // Zone 3 Temperature Control State 4 Start Exhaust Fan
        .5   // Zone 3 Temperature Control State 5 Control to Setpoint
        .6   // Zone 3 Temperature Control State 6 Complete
        .7   // Zone 3 Temperature Control State 7
        .8   // Zone 3 Temperature Control State 8
        .9   // Zone 3 Temperature Control State 9
        .10   // Zone 3 Temperature Control State 10
        .11   // Zone 3 Temperature Control State 11
        .12   // Zone 3 Temperature Control State 12
        .13   // Zone 3 Temperature Control State 13
        .31   // Zone 3 Temperature Control State 31 Manual
   p13r20_status : DINT := 5;   // Zone 3 Temperature Control Sequence Status
   p13r20_timer_fault : TIMER[4];   // Zone 3 Temp Sequence Fault Delay
   p13r20_timer_state_11 : TIMER := (PRE := 5000, ACC := 5001);   // Zone 3 Temp Sequence State 11 Dwell
   p13r20_timer_state_3 : TIMER := (PRE := 1000, ACC := 1024, EN := 1, DN := 1);   // Zone 3 Temperature Control State 3 Dwell
   p13r20_timer_state_4 : TIMER := (PRE := 1000, ACC := 1023, EN := 1, DN := 1);   // Zone 3 Temp Sequence State 4 Dwell
   p13r20_timer_state_7 : TIMER := (PRE := 2000);   // Zone 3 Temp Sequence State 7 Dwell
   p13r20_timer_warning : TIMER[4];   // Zone 3 Temp Sequence Warning Delay
   p13r30 : routine := (comment := -1073741697);   // Zone 3 Temperature Control
        .FAULT.1   // Zone 3 Temperature Control Process Control Hardware High Limit
        .FAULT.2   // Zone 3 Temperature Control Process Control Thermocouple Failure
        .FAULT.3   // Zone 3 Temperature Control Process Control Temperature Spare
        .FAULT.5   // Zone 3 Temperature Control Flame Failure
        .FAULT.6   // Zone 3 Temperature Control Burner Safeties Failure
        .FAULT.7   // Zone 3 Temperature Control Recirculation Fan Speed Fault
        .FAULT.8   // Zone 3 Temperature Control Exhaust Fan Speed Fault
        .FAULT.9   // Zone 3 Temperature Control Access Door Open
        .FAULT.10   // Zone 3 Temperature Control Spare
        .FAULT.11   // Zone 3 Temperature Control
        .FAULT.12   // Zone 3 Temperature Control Spare
        .FAULT.13   // Zone 3 Temperature Control
        .FAULT.14   // Zone 3 Temperature Control
        .WARNING.0   // Zone 3 Temperature Control Control Temperature Deviation
        .WARNING.1   // Zone 3 Temperature Control Process Control Thermocouple 1 Failure
        .WARNING.2   // Zone 3 Temperature Control Process Control Thermocouple 2 Failure
        .WARNING.3   // Zone 3 Temperature Control Control Valve in Manual
        .WARNING.4   // Zone 3 Temperature Control LFL High Limit
        .WARNING.5   // Zone 3 Temperature Control Zone Off
        .WARNING.6   // Zone 3 Temperature Control Fresh Air Filter Dirty
        .WARNING.7   // Zone 3 Temperature Control Zone 3 Filter Dirty
        .WARNING.8   // Zone 3 Temperature Control Recirculation Air Filter Dirty
        .UNACK_FAULT   // Zone 3 Temperature Control Unacknowledged Fault Exists
        .UNACK_WARNING   // Zone 3 Temperature Control Unacknowledged Warning Exists
   p13r30_cv_man_sp : REAL := 80.0;   // Zone 3 Temperature Control Manual Heat Control Valve Setpoint
   p13r30_pb_auto : BOOL;   // Zone 3 Temperature Control PB: Zone Control Auto
   p13r30_pb_manual : BOOL;   // Zone 3 Temperature Control PB: Zone Control Manual
   p13r30_pb_zone_off : BOOL;   // Zone 3 Temperature Control PB: Stop Zone Heat Control
   p13r30_pb_zone_on : BOOL;   // Zone 3 Temperature Control PB: Start Zone Heat Control
   p13r30_permissive_run : BOOL := 1;   // Zone 3 Temperature Control Run Permissive
   p13r30_pid_temp_pv : REAL := 66.3;   // Zone 3 Temperature Control PID Process Value
   p13r30_pid_temp_sp : REAL := 60.0;   // Zone 3 Temperature Control PID Temperature Control Setpoint
   p13r30_pid_temp_sp_error : REAL := 6.300003;   // Zone 3 Temperature Control Setpoint/Process Variable Error (ABS)
   p13r30_pid_temp_sp_last : REAL := 60.0;   // Zone 3 Temperature Control Setpoint Last Scan
   p13r30_request_cool : BOOL := 1;   // Zone 3 Temperature Control Request Cooling
   p13r30_request_deviation_warning : BOOL := 1;   // Zone 3 Temperature Control Request Setpoint Deviation Warning
   p13r30_request_manual : BOOL;   // Zone 3 Temperature Control Request Manual Control
   p13r30_request_PID_shot : BOOL;
   p13r30_temp_deviation_setpoint : DINT := 5;
   p13r30_temp_pid_ctrl : PID := (CTL := -2110745984, EN := 1, CA := 1, NOBC := 1, NOZC := 1, INI := 1, OLH := 1, DVPA := 1, PVHA := 1, SP := 60.0, KP := 10.0, KI := 1.0, MAXS := 1000.0, SO := 100.0, MAXO := 100.0, UPD := 0.1, PV := 65.8, ERR := 5.800003, OUT := 100.0, MAXI := 1000.0, MAXCV := 100.0, MAXTIE := 4095.0, DATA[0] := 97.78058, DATA[1] := 105.28001, DATA[2] := 65.8, DATA[3] := 5.800003, DATA[4] := 60.0, DATA[5] := 0.1, DATA[6] := 1.0, DATA[7] := 1.6, DATA[8] := 10.0, DATA[9] := 1.0, DATA[11] := 10.0, DATA[12] := 1.0, DATA[15] := 1.0, DATA[16] := 0.024420025);   // Zone 3 Temperature Control PID
   p13r30_timer_fault : TIMER[16] := ([0].PRE := 5000, [2].PRE := 1000, [4].PRE := 1000);   // Zone 3 Temperature Control Fault Delay
   p13r30_timer_warning : TIMER[12] := ([0].PRE := 10000, [1].PRE := 1000, [2].PRE := 1000, [3].PRE := 90000, [4].PRE := 1000, [5].PRE := 90000, [6].PRE := 1000, [7].PRE := 1000, [8].PRE := 1000);   // Zone 3 Temperature Control Warning Delay
   p13r30_vfds_ready : BOOL := 1;   // Zone 3 Temperature Control VFDs On
   p13r31 : routine := (comment := -1073741697);   // Zone 3 Exhaust VFD
        .FAULT.0   // Zone 3 Exhaust VFD Drive Fault
        .FAULT.1   // Zone 3 Exhaust VFD Motor Thermistor Not OK
        .FAULT.2   // Zone 3 Exhaust VFD Not Ready
        .FAULT.3   // Zone 3 Exhaust VFD
        .WARNING.0   // Zone 3 Exhaust VFD VFD Stopped While Chamber is Too Hot
        .WARNING.1   // Zone 3 Exhaust VFD Fan Flow Failure
        .WARNING.2   // Zone 3 Exhaust VFD VFD Warning
        .UNACK_FAULT   // Zone 3 Exhaust VFD Unacknowledged Fault Exists
        .UNACK_WARNING   // Zone 3 Exhaust VFD Unacknowledged Warning Exists
   p13r31_pb_start : BOOL;   // Zone 3 Exhaust VFD PB: Start
   p13r31_pb_stop : BOOL;   // Zone 3 Exhaust VFD PB: Stop
   p13r31_request_auto_run : BOOL := 1;   // Zone 3 Exhaust Fan Run Request
   p13r31_request_auto_stop : BOOL := 1;   // Zone 3 Exhaust VFD Request Auto Stop
   p13r31_run_permissive : BOOL := 1;   // Zone 3 Exhaust VFD Run Permissive
   p13r31_timer_fault : TIMER[5] := ([1].PRE := 500);   // Zone 3 Exhaust VFD Fault Timer
   p13r31_timer_warning : TIMER[5] := ([0].PRE := 10000, [1].PRE := 20000, [2].PRE := 500);   // Zone 3 Exhaust VFD Waringing Timer
   p13r31_vfd_stopped : BOOL;   // Zone 3 Exhaust VFD VFD Stopped
   p13r32 : routine := (comment := -536870849);   // Zone 3 Recirc VFD
        .FAULT.0   // Zone 3 Recirc VFD Drive Fault
        .FAULT.1   // Zone 3 Recirc VFD Motor Thermistor Not OK
        .FAULT.2   // Zone 3 Recirc VFD Not Ready
        .FAULT.3   // Zone 3 Supply VFD
        .WARNING.0   // Zone 3 Recirc VFD VFD Stopped While Chamber is Too Hot
        .WARNING.1   // Zone 3 Recirc VFD Fan Flow Failure
        .WARNING.2   // Zone 3 Recirc VFD VFD Warning
        .UNACK_FAULT   // Zone 3 Recirc VFD Unacknowledged Fault Exists
        .UNACK_WARNING   // Zone 3 Recirc VFD Unacknowledged Warning Exists
   p13r32_pb_start : BOOL;   // Zone 3 Recirc VFD PB: Start
   p13r32_pb_stop : BOOL;   // Zone 3 Recirc VFD PB: Stop
   p13r32_request_auto_run : BOOL := 1;   // Zone 3 Recirc Fan Run Request
   p13r32_request_auto_stop : BOOL;   // Zone 3 Recirc VFD Request Auto Stop
   p13r32_run_permissive : BOOL := 1;   // Zone 3 Recirc VFD Run Permissive
   p13r32_timer_fault : TIMER[5] := ([1].PRE := 500);   // Zone 3 Recirc VFD Fault Timer
   p13r32_timer_warning : TIMER[5] := ([0].PRE := 10000, [1].PRE := 20000, [2].PRE := 20000);   // Zone 3 Supply VFD Warning Timer
   p13r32_vfd_stopped : BOOL;   // Zone 3 Recirc VFD VFD Stopped
   p19_ai_prs : REAL := 14.765242;   // Advanced Cooling Analog Input Pressure [PSI]
   p19_ai_tc01 : REAL := 59.5;   // Advanced Cooling Analog Input Control Temperature 1
   p19_ao_cv : REAL := 12.04493;   // Advanced Cooling Analog Output Control Valve
   p19_ao_prs_cv : REAL := 1.5767791;   // Advanced Cooling Pressure Control AO: Control Value
   p19_di_pump : BOOL := 1;
   p19_di_tc01_bo : BOOL;   // Advanced Cooling Digital Input Control Thermocouple 1 Failure
   p19_di_tc02_bo : BOOL := 1;   // Advanced Cooling Digital Input Control Thermocouple 2 Failure
   p19_dint_to_hmi : DINT[16] := ([0] := 589840, [1] := 32769, [5] := 16382);
        [0].0   // Advanced Cooling Dint to HMI
        [0].1   // Advanced Cooling Dint to HMI
        [0].2   // Advanced Cooling Dint to HMI
        [0].3   // Advanced Cooling Dint to HMI
        [0].4   // Advanced Cooling Dint to HMI Pump Request Auto Run
        [0].5   // Advanced Cooling Dint to HMI
        [0].6   // Advanced Cooling Dint to HMI
        [0].7   // Advanced Cooling Dint to HMI
        [0].8   // Advanced Cooling Dint to HMI
        [0].9   // Advanced Cooling Dint to HMI
        [0].10   // Advanced Cooling Dint to HMI
        [0].11   // Advanced Cooling Dint to HMI
        [0].12   // Advanced Cooling Dint to HMI
        [0].13   // Advanced Cooling Dint to HMI
        [0].14   // Advanced Cooling Dint to HMI
        [0].15   // Advanced Cooling Dint to HMI
        [0].16   // Advanced Cooling Dint to HMI Temperature Control Request Cool
        [0].17   // Advanced Cooling Dint to HMI Temperature Control Request Heat
        [0].18   // Advanced Cooling Dint to HMI Temperature Control Request Manual Control
        [0].19   // Advanced Cooling Dint to HMI Temperature Control Request Auto Control
        [0].20   // Advanced Cooling Dint to HMI
        [0].21   // Advanced Cooling Dint to HMI
        [0].22   // Advanced Cooling Dint to HMI
        [0].23   // Advanced Cooling Dint to HMI
        [0].24   // Advanced Cooling Dint to HMI
        [0].25   // Advanced Cooling Dint to HMI
        [0].26   // Advanced Cooling Dint to HMI
        [0].27   // Advanced Cooling Dint to HMI
        [0].28   // Advanced Cooling Dint to HMI
        [0].29   // Advanced Cooling Dint to HMI
        [0].30   // Advanced Cooling Dint to HMI
        [0].31   // Advanced Cooling Dint to HMI
        [1].0   // Advanced Cooling Dint to HMI
        [1].1   // Advanced Cooling Dint to HMI
        [1].2   // Advanced Cooling Dint to HMI
        [1].3   // Advanced Cooling Dint to HMI
        [1].4   // Advanced Cooling Dint to HMI
        [1].5   // Advanced Cooling Dint to HMI
        [1].6   // Advanced Cooling Dint to HMI
        [1].7   // Advanced Cooling Dint to HMI
        [1].8   // Advanced Cooling Dint to HMI
        [1].9   // Advanced Cooling Dint to HMI
        [1].10   // Advanced Cooling Dint to HMI
        [1].11   // Advanced Cooling Dint to HMI
        [1].12   // Advanced Cooling Dint to HMI
        [1].13   // Advanced Cooling Dint to HMI
        [1].14   // Advanced Cooling Dint to HMI Control Thermocouple 1 Failure
        [1].15   // Advanced Cooling Dint to HMI Control Thermocouple 2 Failure
        [2].0   // Advanced Cooling Dint to HMI Alarms A00:
        [2].1   // Advanced Cooling Dint to HMI Alarms A01:
        [2].2   // Advanced Cooling Dint to HMI Alarms A02: Process Control Thermocouple Failure
        [2].3   // Advanced Cooling Dint to HMI Alarms A03:
        [2].4   // Advanced Cooling Dint to HMI Alarms A04:
        [2].5   // Advanced Cooling Dint to HMI Alarms A05:
        [2].6   // Advanced Cooling Dint to HMI Alarms A06:
        [2].7   // Advanced Cooling Dint to HMI Alarms A07:
        [2].8   // Advanced Cooling Dint to HMI Alarms A08:
        [2].9   // Advanced Cooling Dint to HMI Alarms A09:
        [2].10   // Advanced Cooling Dint to HMI Alarms A10:
        [2].11   // Advanced Cooling Dint to HMI Alarms A11:
        [2].12   // Advanced Cooling Dint to HMI Alarms A12:
        [2].13   // Advanced Cooling Dint to HMI Alarms A13:
        [2].14   // Advanced Cooling Dint to HMI Alarms A14:
        [2].15   // Advanced Cooling Dint to HMI Alarms A15:
        [2].16   // Advanced Cooling Dint to HMI Alarms A16: Low Pump Pressure
        [2].17   // Advanced Cooling Dint to HMI Alarms A17:
        [2].18   // Advanced Cooling Dint to HMI Alarms A18:
        [2].19   // Advanced Cooling Dint to HMI Alarms A19:
        [2].20   // Advanced Cooling Dint to HMI Alarms A20:
        [2].21   // Advanced Cooling Dint to HMI Alarms A21:
        [2].22   // Advanced Cooling Dint to HMI Alarms A22:
        [2].23   // Advanced Cooling Dint to HMI Alarms A23:
        [2].28   // Advanced Cooling Dint to HMI Alarms A28:
        [2].29   // Advanced Cooling Dint to HMI Alarms A29:
        [2].30   // Advanced Cooling Dint to HMI Alarms A30:
        [2].31   // Advanced Cooling Dint to HMI Alarms A31:
        [4].0   // Advanced Cooling Warning W00: Temperature Deviation
        [4].1   // Advanced Cooling Warning W01: Control Thermocouple 1 Failure
        [4].2   // Advanced Cooling Warning W02: Control Thermocouple 2 Failure
        [4].3   // Advanced Cooling Warning W03: Temperature Control in Manual
        [4].4   // Advanced Cooling Warning W04:
        [4].5   // Advanced Cooling Warning W05:
        [4].6   // Advanced Cooling Warning W06:
        [4].7   // Advanced Cooling Warning W07:
        [4].8   // Advanced Cooling Warning W08:
        [4].9   // Advanced Cooling Warning W09:
        [4].10   // Advanced Cooling Warning W10:
        [4].11   // Advanced Cooling Warning W11:
        [4].12   // Advanced Cooling Warning W12:
        [4].13   // Advanced Cooling Warning W13:
        [4].14   // Advanced Cooling Warning W14:
        [4].15   // Advanced Cooling Warning W15:
        [4].16   // Advanced Cooling Warning W16: Pump Off
        [4].17   // Advanced Cooling Warning W17:
        [4].18   // Advanced Cooling Warning W18:
        [4].19   // Advanced Cooling Warning W19:
   p19_do_pump : BOOL := 1;   // Advanced Cooling Digital Output Enable Pump
   p19_flow_input_max : REAL := 100.0;
   p19_flow_input_min : REAL;
   p19_flow_output_max : REAL := 30840.0;
   p19_flow_output_min : REAL;
   p19_param_pid1_ff : REAL;
   p19_param_pid1_kd : REAL;
   p19_param_pid1_ki : REAL;
   p19_param_pid1_kp : REAL;
   p19_param_pid2_ff : REAL;
   p19_param_pid2_kd : REAL;
   p19_param_pid2_ki : REAL := 1.0;
